C07305=1131.098,83.336,-54.639,179.925,7.711,149.479
C07306=1131.094,83.586,-54.656,179.926,7.715,149.480
C07307=1131.089,83.835,-54.674,179.927,7.718,149.480
C07308=1131.084,84.085,-54.691,179.929,7.722,149.481
C07309=1131.079,84.334,-54.709,179.930,7.726,149.481
C07310=1131.075,84.583,-54.727,179.932,7.730,149.482
C07311=1131.069,84.833,-54.744,179.932,7.734,149.482
C07312=1131.065,85.082,-54.762,179.934,7.738,149.483
C07313=1131.059,85.332,-54.779,179.935,7.742,149.483
C07314=1131.055,85.580,-54.796,179.937,7.745,149.483
C07315=1131.050,85.830,-54.814,179.938,7.749,149.484
C07316=1131.045,86.079,-54.832,179.939,7.753,149.485
C07317=1131.040,86.329,-54.850,179.941,7.757,149.485
C07318=1131.035,86.578,-54.867,179.942,7.761,149.486
C07319=1131.031,86.827,-54.884,179.943,7.765,149.486
C07320=1131.026,87.076,-54.902,179.945,7.769,149.486
C07321=1131.021,87.326,-54.920,179.947,7.773,149.487
C07322=1131.016,87.575,-54.938,179.947,7.776,149.487
C07323=1131.011,87.825,-54.955,179.949,7.780,149.488
C07324=1131.006,88.074,-54.973,179.950,7.784,149.488
C07325=1131.001,88.324,-54.991,179.952,7.788,149.489
C07326=1130.996,88.572,-55.008,179.954,7.792,149.489
C07327=1130.992,88.822,-55.026,179.955,7.796,149.490
C07328=1130.984,89.194,-55.053,179.957,7.802,149.490
C07329=1130.977,89.567,-55.079,179.959,7.808,149.491
C07330=1130.969,89.939,-55.106,179.962,7.814,149.492
C07331=1130.962,90.311,-55.132,179.964,7.819,149.492
C07332=1130.958,90.561,-55.150,179.966,7.823,149.493
C07333=1130.952,90.811,-55.167,179.967,7.827,149.493
C07334=1130.948,91.060,-55.185,179.969,7.831,149.494
C07335=1130.943,91.309,-55.203,179.971,7.835,149.494
C07336=1130.938,91.558,-55.221,179.972,7.839,149.495
C07337=1130.933,91.807,-55.239,179.974,7.843,149.495
C07338=1130.928,92.056,-55.257,179.975,7.847,149.495
C07339=1130.923,92.306,-55.275,179.977,7.851,149.496
C07340=1130.918,92.555,-55.293,179.979,7.854,149.496
C07341=1130.913,92.804,-55.311,179.980,7.858,149.497
C07342=1130.908,93.054,-55.329,179.982,7.863,149.497
C07343=1130.904,93.304,-55.347,179.984,7.867,149.498
C07344=1130.899,93.553,-55.365,179.986,7.871,149.498
C07345=1130.894,93.802,-55.383,179.987,7.875,149.498
C07346=1130.889,94.051,-55.401,179.989,7.879,149.499
C07347=1130.884,94.300,-55.419,179.990,7.882,149.499
C07348=1130.878,94.550,-55.437,179.992,7.886,149.500
C07349=1130.873,94.799,-55.455,179.994,7.891,149.500
C07350=1130.869,95.049,-55.474,179.996,7.895,149.500
C07351=1130.864,95.298,-55.492,179.998,7.898,149.501
C07352=1130.859,95.547,-55.510,180.000,7.902,149.501
C07353=1130.854,95.796,-55.528,-179.999,7.906,149.502
C07354=1130.850,96.045,-55.546,-179.997,7.911,149.502
C07355=1130.845,96.294,-55.564,-179.995,7.914,149.502
C07356=1130.841,96.544,-55.583,-179.993,7.918,149.503
C07357=1130.835,96.793,-55.601,-179.991,7.922,149.503
C07358=1130.830,97.043,-55.619,-179.989,7.927,149.503
C07359=1130.825,97.292,-55.637,-179.987,7.930,149.504
C07360=1130.820,97.541,-55.655,-179.986,7.934,149.504
C07361=1130.816,97.791,-55.673,-179.984,7.938,149.505
C07362=1130.811,98.039,-55.692,-179.981,7.942,149.505
C07363=1130.806,98.289,-55.711,-179.980,7.946,149.505
C07364=1130.801,98.538,-55.729,-179.978,7.950,149.506
C07365=1130.796,98.788,-55.747,-179.975,7.954,149.506
C07366=1130.791,99.037,-55.765,-179.974,7.958,149.506
C07367=1130.787,99.286,-55.784,-179.972,7.962,149.507
C07368=1130.781,99.535,-55.802,-179.969,7.967,149.507
C07369=1130.777,99.785,-55.821,-179.968,7.970,149.507
C07370=1130.772,100.034,-55.839,-179.966,7.974,149.508
C07371=1130.767,100.283,-55.857,-179.964,7.979,149.508
C07372=1130.762,100.532,-55.876,-179.962,7.982,149.508
C07373=1130.757,100.782,-55.894,-179.959,7.987,149.509
C07374=1130.753,101.031,-55.913,-179.957,7.990,149.509
C07375=1130.747,101.280,-55.932,-179.956,7.994,149.509
C07376=1130.743,101.530,-55.950,-179.953,7.998,149.509
C07377=1130.738,101.779,-55.969,-179.951,8.002,149.510
C07378=1130.733,102.028,-55.987,-179.949,8.007,149.510
C07379=1130.728,102.277,-56.005,-179.947,8.010,149.510
C07380=1130.724,102.492,-56.022,-179.945,8.014,149.511
C07381=1130.720,102.707,-56.038,-179.943,8.018,149.511
C07382=1130.716,102.923,-56.053,-179.941,8.021,149.511
C07383=1130.711,103.137,-56.070,-179.939,8.025,149.511
C07384=1130.707,103.352,-56.085,-179.937,8.028,149.512
C07385=1130.703,103.567,-56.102,-179.935,8.031,149.512
C07386=1130.699,103.782,-56.118,-179.933,8.034,149.512
C07387=1130.695,103.997,-56.134,-179.932,8.038,149.512
C07388=1130.690,104.246,-56.154,-179.929,8.042,149.513
C07389=1130.685,104.495,-56.171,-179.927,8.046,149.513
C07390=1130.681,104.745,-56.191,-179.924,8.050,149.513
C07391=1130.675,104.994,-56.209,-179.923,8.054,149.514
C07392=1130.670,105.243,-56.228,-179.920,8.058,149.514
C07393=1130.665,105.493,-56.247,-179.918,8.062,149.514
C07394=1130.661,105.741,-56.265,-179.915,8.066,149.514
C07395=1130.656,105.992,-56.284,-179.912,8.070,149.514
C07396=1130.651,106.240,-56.303,-179.910,8.074,149.515
C07397=1130.646,106.490,-56.323,-179.908,8.078,149.515
C07398=1130.642,106.739,-56.341,-179.906,8.082,149.515
C07399=1130.636,106.988,-56.360,-179.903,8.086,149.516
C07400=1130.632,107.237,-56.379,-179.901,8.091,149.516
C07401=1130.627,107.487,-56.398,-179.899,8.094,149.516
C07402=1130.623,107.736,-56.417,-179.896,8.098,149.516
C07403=1130.617,107.985,-56.436,-179.894,8.102,149.516
C07404=1130.613,108.235,-56.454,-179.891,8.106,149.517
C07405=1130.608,108.483,-56.474,-179.888,8.110,149.517
C07406=1130.603,108.733,-56.493,-179.886,8.114,149.517
C07407=1130.598,108.982,-56.512,-179.883,8.118,149.517
C07408=1130.593,109.232,-56.531,-179.881,8.122,149.517
C07409=1130.588,109.480,-56.550,-179.879,8.126,149.517
C07410=1130.584,109.730,-56.569,-179.876,8.130,149.518
C07411=1130.579,109.978,-56.588,-179.873,8.134,149.518
C07412=1130.574,110.228,-56.608,-179.871,8.139,149.518
C07413=1130.569,110.477,-56.627,-179.868,8.142,149.518
C07414=1130.565,110.727,-56.645,-179.865,8.146,149.518
C07415=1130.559,110.976,-56.665,-179.863,8.149,149.519
C07416=1130.555,111.225,-56.684,-179.861,8.153,149.519
C07417=1130.550,111.474,-56.703,-179.859,8.156,149.519
C07418=1130.545,111.723,-56.723,-179.858,8.160,149.519
C07419=1130.540,111.972,-56.742,-179.856,8.164,149.520
C07420=1130.535,112.222,-56.762,-179.853,8.167,149.520
C07421=1130.531,112.471,-56.781,-179.851,8.171,149.520
C07422=1130.526,112.720,-56.800,-179.849,8.174,149.520
C07423=1130.521,112.969,-56.820,-179.848,8.178,149.521
C07424=1130.517,113.218,-56.838,-179.846,8.182,149.521
C07425=1130.512,113.468,-56.858,-179.844,8.185,149.521
C07426=1130.506,113.716,-56.877,-179.842,8.189,149.521
C07427=1130.502,113.966,-56.897,-179.839,8.192,149.522
C07428=1130.497,114.216,-56.916,-179.838,8.196,149.522
C07429=1130.492,114.464,-56.935,-179.836,8.200,149.522
C07430=1130.488,114.714,-56.955,-179.834,8.203,149.523
C07431=1130.482,114.963,-56.974,-179.832,8.207,149.523
C07432=1130.478,115.212,-56.994,-179.830,8.210,149.523
C07433=1130.473,115.462,-57.013,-179.828,8.214,149.523
C07434=1130.468,115.710,-57.032,-179.826,8.217,149.524
C07435=1130.463,115.960,-57.052,-179.824,8.221,149.524
C07436=1130.459,116.175,-57.069,-179.822,8.224,149.524
C07437=1130.455,116.389,-57.086,-179.821,8.226,149.524
C07438=1130.451,116.604,-57.103,-179.819,8.230,149.524
C07439=1130.447,116.820,-57.120,-179.817,8.233,149.525
C07440=1130.442,117.034,-57.136,-179.816,8.235,149.525
C07441=1130.438,117.249,-57.153,-179.814,8.239,149.525
C07442=1130.434,117.464,-57.170,-179.813,8.241,149.525
C07443=1130.430,117.679,-57.187,-179.811,8.244,149.526
C07444=1130.425,117.928,-57.207,-179.809,8.248,149.526
C07445=1130.421,118.176,-57.226,-179.807,8.251,149.526
C07446=1130.416,118.426,-57.246,-179.805,8.255,149.526
C07447=1130.411,118.675,-57.266,-179.803,8.259,149.527
C07448=1130.407,118.925,-57.285,-179.801,8.262,149.527
C07449=1130.402,119.173,-57.305,-179.800,8.265,149.527
C07450=1130.397,119.423,-57.325,-179.798,8.268,149.527
C07451=1130.392,119.672,-57.345,-179.796,8.272,149.528
C07452=1130.387,119.920,-57.365,-179.794,8.276,149.528
C07453=1130.382,120.170,-57.384,-179.792,8.279,149.528
C07454=1130.378,120.420,-57.404,-179.790,8.283,149.528
C07455=1130.373,120.669,-57.424,-179.788,8.285,149.529
C07456=1130.368,120.917,-57.444,-179.786,8.289,149.529
C07457=1130.363,121.167,-57.463,-179.785,8.293,149.529
C07458=1130.359,121.416,-57.484,-179.783,8.296,149.530
C07459=1130.354,121.666,-57.503,-179.781,8.300,149.530
C07460=1130.349,121.914,-57.522,-179.779,8.302,149.530
C07461=1130.344,122.163,-57.543,-179.777,8.306,149.530
C07462=1130.339,122.413,-57.563,-179.775,8.309,149.530
C07463=1130.335,122.662,-57.583,-179.773,8.313,149.531
C07464=1130.330,122.911,-57.603,-179.772,8.316,149.531
C07465=1130.325,123.160,-57.622,-179.770,8.320,149.531
C07466=1130.320,123.409,-57.642,-179.768,8.323,149.532
C07467=1130.316,123.659,-57.662,-179.766,8.327,149.532
C07468=1130.311,123.908,-57.682,-179.765,8.330,149.532
C07469=1130.307,124.157,-57.702,-179.763,8.333,149.532
C07470=1130.301,124.406,-57.722,-179.761,8.337,149.533
C07471=1130.297,124.655,-57.742,-179.759,8.339,149.533
C07472=1130.292,124.904,-57.763,-179.758,8.343,149.533
C07473=1130.287,125.154,-57.782,-179.756,8.347,149.533
C07474=1130.282,125.403,-57.803,-179.753,8.350,149.534
C07475=1130.278,125.652,-57.823,-179.752,8.353,149.534
C07476=1130.273,125.901,-57.842,-179.750,8.356,149.534
C07477=1130.268,126.150,-57.863,-179.748,8.360,149.535
C07478=1130.263,126.399,-57.882,-179.747,8.363,149.535
C07479=1130.259,126.648,-57.903,-179.745,8.366,149.535
C07480=1130.254,126.897,-57.924,-179.743,8.370,149.535
C07481=1130.249,127.147,-57.943,-179.742,8.373,149.536
C07482=1130.245,127.396,-57.964,-179.740,8.377,149.536
C07483=1130.239,127.645,-57.983,-179.738,8.380,149.536
C07484=1130.235,127.894,-58.003,-179.736,8.383,149.536
C07485=1130.230,128.143,-58.024,-179.735,8.387,149.537
C07486=1130.225,128.393,-58.044,-179.732,8.390,149.537
C07487=1130.220,128.642,-58.064,-179.731,8.393,149.537
C07488=1130.216,128.891,-58.085,-179.729,8.397,149.538
C07489=1130.212,129.139,-58.105,-179.727,8.400,149.538
C07490=1130.206,129.389,-58.125,-179.726,8.403,149.538
C07491=1130.202,129.638,-58.146,-179.724,8.406,149.538
C07492=1130.197,129.852,-58.163,-179.722,8.409,149.539
C07493=1130.193,130.067,-58.180,-179.721,8.412,149.539
C07494=1130.189,130.282,-58.198,-179.720,8.415,149.539
C07495=1130.185,130.497,-58.216,-179.718,8.418,149.539
C07496=1130.181,130.712,-58.233,-179.717,8.420,149.540
C07497=1130.177,130.927,-58.251,-179.715,8.424,149.540
C07498=1130.173,131.141,-58.268,-179.713,8.427,149.540
C07499=1130.169,131.356,-58.285,-179.712,8.429,149.540
C07500=1130.164,131.605,-58.306,-179.711,8.432,149.541
C07501=1130.159,131.854,-58.327,-179.709,8.436,149.541
C07502=1130.155,132.103,-58.347,-179.708,8.439,149.541
C07503=1130.150,132.352,-58.368,-179.706,8.443,149.542
C07504=1130.145,132.602,-58.388,-179.704,8.446,149.542
C07505=1130.140,132.851,-58.408,-179.702,8.449,149.542
C07506=1130.136,133.100,-58.429,-179.701,8.453,149.543
C07507=1130.131,133.349,-58.449,-179.699,8.455,149.543
C07508=1130.126,133.598,-58.470,-179.697,8.459,149.543
C07509=1130.122,133.847,-58.490,-179.696,8.462,149.543
C07510=1130.117,134.096,-58.511,-179.694,8.465,149.544
C07511=1130.112,134.345,-58.532,-179.693,8.469,149.544
C07512=1130.107,134.595,-58.553,-179.691,8.472,149.544
C07513=1130.102,134.843,-58.573,-179.689,8.475,149.544
C07514=1130.098,135.092,-58.593,-179.688,8.479,149.545
C07515=1130.093,135.342,-58.614,-179.686,8.482,149.545
C07516=1130.088,135.591,-58.635,-179.685,8.485,149.546
C07517=1130.083,135.840,-58.656,-179.683,8.489,149.546
C07518=1130.079,136.089,-58.676,-179.681,8.491,149.546
C07519=1130.074,136.338,-58.697,-179.680,8.495,149.546
C07520=1130.069,136.587,-58.717,-179.678,8.498,149.547
C07521=1130.065,136.836,-58.738,-179.677,8.502,149.547
C07522=1130.060,137.085,-58.759,-179.675,8.505,149.547
C07523=1130.055,137.334,-58.779,-179.674,8.508,149.548
C07524=1130.050,137.583,-58.800,-179.672,8.511,149.548
C07525=1130.046,137.832,-58.820,-179.670,8.515,149.548
C07526=1130.041,138.082,-58.842,-179.669,8.518,149.549
C07527=1130.037,138.331,-58.862,-179.667,8.521,149.549
C07528=1130.031,138.581,-58.883,-179.666,8.524,149.549
C07529=1130.027,138.830,-58.903,-179.664,8.528,149.550
C07530=1130.022,139.078,-58.925,-179.663,8.531,149.550
C07531=1130.018,139.327,-58.945,-179.661,8.534,149.550
C07532=1130.012,139.576,-58.966,-179.660,8.537,149.551
C07533=1130.008,139.825,-58.987,-179.658,8.541,149.551
C07534=1130.003,140.075,-59.008,-179.657,8.544,149.551
C07535=1129.998,140.324,-59.028,-179.655,8.548,149.552
C07536=1129.994,140.572,-59.050,-179.654,8.551,149.552
C07537=1129.989,140.822,-59.071,-179.652,8.554,149.552
C07538=1129.984,141.071,-59.091,-179.651,8.557,149.553
C07539=1129.979,141.320,-59.112,-179.650,8.560,149.553
C07540=1129.975,141.569,-59.133,-179.647,8.564,149.553
C07541=1129.970,141.818,-59.155,-179.646,8.567,149.554
C07542=1129.966,142.067,-59.175,-179.645,8.571,149.554
C07543=1129.960,142.316,-59.196,-179.643,8.573,149.554
C07544=1129.956,142.566,-59.217,-179.642,8.577,149.555
C07545=1129.952,142.814,-59.238,-179.640,8.580,149.555
C07546=1129.947,143.064,-59.259,-179.639,8.584,149.555
C07547=1129.941,143.313,-59.280,-179.638,8.587,149.556
C07548=1129.938,143.527,-59.298,-179.636,8.590,149.556
C07549=1129.933,143.742,-59.316,-179.635,8.593,149.557
C07550=1129.930,143.957,-59.334,-179.634,8.595,149.557
C07551=1129.926,144.171,-59.353,-179.632,8.598,149.557
C07552=1129.922,144.385,-59.371,-179.631,8.601,149.557
C07553=1129.918,144.600,-59.389,-179.630,8.604,149.558
C07554=1129.913,144.815,-59.408,-179.629,8.607,149.558
C07555=1129.909,145.030,-59.426,-179.627,8.610,149.558
C07556=1129.904,145.279,-59.446,-179.625,8.613,149.559
C07557=1129.900,145.528,-59.469,-179.623,8.618,149.559
C07558=1129.896,145.777,-59.489,-179.619,8.621,149.559
C07559=1129.890,146.026,-59.510,-179.617,8.626,149.559
C07560=1129.886,146.275,-59.532,-179.614,8.630,149.559
C07561=1129.881,146.524,-59.552,-179.611,8.634,149.559
C07562=1129.877,146.773,-59.574,-179.609,8.637,149.559
C07563=1129.872,147.023,-59.595,-179.606,8.642,149.560
C07564=1129.867,147.271,-59.617,-179.603,8.646,149.560
C07565=1129.862,147.520,-59.637,-179.600,8.650,149.560
C07566=1129.858,147.770,-59.659,-179.598,8.653,149.560
C07567=1129.853,148.019,-59.680,-179.595,8.657,149.560
C07568=1129.848,148.267,-59.702,-179.592,8.661,149.560
C07569=1129.843,148.517,-59.723,-179.589,8.666,149.561
C07570=1129.839,148.766,-59.745,-179.587,8.669,149.561
C07571=1129.834,149.014,-59.766,-179.584,8.673,149.561
C07572=1129.829,149.264,-59.787,-179.582,8.677,149.561
C07573=1129.825,149.513,-59.809,-179.579,8.680,149.561
C07574=1129.820,149.762,-59.830,-179.576,8.685,149.561
C07575=1129.815,150.011,-59.851,-179.573,8.689,149.561
C07576=1129.811,150.260,-59.874,-179.571,8.692,149.562
C07577=1129.806,150.509,-59.895,-179.568,8.696,149.562
C07578=1129.801,150.758,-59.916,-179.566,8.699,149.562
C07579=1129.797,151.007,-59.938,-179.563,8.703,149.562
C07580=1129.792,151.256,-59.959,-179.560,8.708,149.562
C07581=1129.787,151.504,-59.981,-179.557,8.711,149.562
C07582=1129.783,151.754,-60.002,-179.555,8.715,149.563
C07583=1129.778,152.003,-60.024,-179.552,8.718,149.563
C07584=1129.773,152.252,-60.046,-179.550,8.722,149.563
C07585=1129.769,152.501,-60.068,-179.547,8.725,149.563
C07586=1129.764,152.750,-60.089,-179.544,8.730,149.563
C07587=1129.759,153.000,-60.111,-179.542,8.733,149.563
C07588=1129.755,153.248,-60.132,-179.539,8.737,149.563
C07589=1129.750,153.497,-60.154,-179.537,8.740,149.563
C07590=1129.745,153.746,-60.176,-179.534,8.744,149.564
C07591=1129.741,153.995,-60.198,-179.531,8.747,149.564
C07592=1129.736,154.244,-60.220,-179.528,8.751,149.564
C07593=1129.731,154.493,-60.242,-179.526,8.755,149.564
C07594=1129.727,154.741,-60.263,-179.523,8.759,149.564
C07595=1129.722,154.991,-60.285,-179.521,8.762,149.564
C07596=1129.717,155.240,-60.308,-179.518,8.765,149.564
C07597=1129.712,155.489,-60.330,-179.515,8.769,149.564
C07598=1129.708,155.738,-60.351,-179.513,8.773,149.564
C07599=1129.703,155.987,-60.373,-179.510,8.777,149.564
C07600=1129.698,156.236,-60.395,-179.508,8.780,149.565
C07601=1129.694,156.485,-60.417,-179.505,8.783,149.565
C07602=1129.689,156.734,-60.439,-179.502,8.787,149.565
C07603=1129.685,156.983,-60.461,-179.500,8.791,149.565
C07604=1129.681,157.198,-60.479,-179.498,8.794,149.565
C07605=1129.676,157.412,-60.498,-179.496,8.796,149.565
C07606=1129.672,157.626,-60.517,-179.494,8.799,149.565
C07607=1129.669,157.841,-60.537,-179.491,8.803,149.565
C07608=1129.665,158.056,-60.555,-179.489,8.806,149.565
C07609=1129.660,158.270,-60.574,-179.487,8.808,149.565
C07610=1129.657,158.485,-60.594,-179.485,8.812,149.566
C07611=1129.653,158.699,-60.613,-179.482,8.815,149.566
C07612=1129.647,158.948,-60.635,-179.479,8.818,149.566
C07613=1129.643,159.198,-60.657,-179.477,8.821,149.566
C07614=1129.638,159.446,-60.679,-179.475,8.824,149.566
C07615=1129.634,159.695,-60.701,-179.472,8.828,149.566
C07616=1129.629,159.945,-60.724,-179.469,8.831,149.566
C07617=1129.624,160.193,-60.746,-179.467,8.835,149.566
C07618=1129.620,160.443,-60.768,-179.465,8.838,149.566
C07619=1129.615,160.691,-60.790,-179.462,8.841,149.566
C07620=1129.610,160.940,-60.813,-179.460,8.845,149.566
C07621=1129.606,161.190,-60.835,-179.457,8.848,149.567
C07622=1129.601,161.438,-60.857,-179.454,8.851,149.567
C07623=1129.597,161.687,-60.880,-179.452,8.855,149.567
C07624=1129.592,161.936,-60.902,-179.450,8.858,149.567
C07625=1129.587,162.185,-60.924,-179.447,8.861,149.567
C07626=1129.583,162.434,-60.947,-179.445,8.864,149.567
C07627=1129.578,162.683,-60.969,-179.443,8.868,149.567
C07628=1129.574,162.932,-60.991,-179.439,8.872,149.567
C07629=1129.568,163.181,-61.014,-179.437,8.875,149.567
C07630=1129.564,163.430,-61.036,-179.434,8.878,149.567
C07631=1129.560,163.679,-61.059,-179.432,8.881,149.567
C07632=1129.555,163.928,-61.081,-179.430,8.884,149.567
C07633=1129.551,164.176,-61.104,-179.427,8.888,149.568
C07634=1129.546,164.426,-61.126,-179.425,8.891,149.568
C07635=1129.541,164.675,-61.148,-179.423,8.894,149.568
C07636=1129.537,164.923,-61.171,-179.420,8.897,149.568
C07637=1129.532,165.173,-61.193,-179.418,8.900,149.568
C07638=1129.527,165.421,-61.216,-179.415,8.903,149.568
C07639=1129.522,165.670,-61.239,-179.413,8.907,149.568
C07640=1129.518,165.919,-61.261,-179.410,8.910,149.568
C07641=1129.513,166.168,-61.285,-179.408,8.913,149.568
C07642=1129.509,166.417,-61.306,-179.405,8.916,149.568
C07643=1129.505,166.666,-61.329,-179.403,8.919,149.568
C07644=1129.500,166.915,-61.352,-179.401,8.923,149.568
C07645=1129.495,167.163,-61.374,-179.398,8.926,149.569
C07646=1129.490,167.412,-61.397,-179.396,8.929,149.569
C07647=1129.485,167.662,-61.420,-179.393,8.932,149.569
C07648=1129.481,167.911,-61.443,-179.391,8.936,149.569
C07649=1129.476,168.160,-61.465,-179.389,8.938,149.569
C07650=1129.472,168.408,-61.488,-179.387,8.941,149.569
C07651=1129.467,168.657,-61.511,-179.384,8.944,149.569
C07652=1129.463,168.906,-61.534,-179.382,8.948,149.569
C07653=1129.458,169.155,-61.556,-179.380,8.951,149.569
C07654=1129.454,169.404,-61.579,-179.377,8.954,149.569
C07655=1129.449,169.653,-61.602,-179.375,8.957,149.569
C07656=1129.444,169.903,-61.625,-179.372,8.961,149.569
C07657=1129.439,170.151,-61.648,-179.371,8.963,149.570
C07658=1129.435,170.400,-61.671,-179.368,8.966,149.570
C07659=1129.431,170.648,-61.694,-179.365,8.969,149.570
C07660=1129.426,170.863,-61.713,-179.364,8.972,149.570
C07661=1129.422,171.078,-61.733,-179.361,8.975,149.570
C07662=1129.418,171.292,-61.753,-179.360,8.977,149.570
C07663=1129.414,171.507,-61.773,-179.358,8.980,149.570
C07664=1129.410,171.721,-61.792,-179.355,8.983,149.570
C07665=1129.406,171.935,-61.812,-179.354,8.985,149.570
C07666=1129.402,172.149,-61.832,-179.352,8.988,149.570
C07667=1129.398,172.364,-61.852,-179.350,8.990,149.570
C07668=1129.394,172.613,-61.875,-179.347,8.993,149.570
C07669=1129.389,172.862,-61.898,-179.345,8.997,149.571
C07670=1129.385,173.111,-61.921,-179.343,9.000,149.571
C07671=1129.379,173.360,-61.944,-179.341,9.002,149.571
C07672=1129.375,173.609,-61.967,-179.338,9.005,149.571
C07673=1129.371,173.858,-61.990,-179.336,9.009,149.571
C07674=1129.366,174.107,-62.014,-179.334,9.011,149.571
C07675=1129.362,174.355,-62.036,-179.332,9.014,149.571
C07676=1129.357,174.604,-62.060,-179.330,9.018,149.571
C07677=1129.353,174.853,-62.083,-179.327,9.021,149.571
C07678=1129.347,175.102,-62.106,-179.325,9.023,149.571
C07679=1129.343,175.350,-62.129,-179.323,9.026,149.571
C07680=1129.339,175.599,-62.152,-179.321,9.030,149.571
C07681=1129.334,175.848,-62.176,-179.319,9.032,149.572
C07682=1129.329,176.098,-62.199,-179.316,9.035,149.572
C07683=1129.325,176.347,-62.222,-179.314,9.038,149.572
C07684=1129.321,176.595,-62.245,-179.312,9.041,149.572
C07685=1129.316,176.844,-62.268,-179.310,9.044,149.572
C07686=1129.311,177.093,-62.292,-179.308,9.047,149.572
C07687=1129.307,177.342,-62.315,-179.306,9.050,149.572
C07688=1129.302,177.591,-62.339,-179.303,9.053,149.572
C07689=1129.298,177.839,-62.362,-179.302,9.056,149.572
C07690=1129.293,178.089,-62.385,-179.299,9.059,149.572
C07691=1129.288,178.337,-62.408,-179.297,9.062,149.573
C07692=1129.283,178.586,-62.432,-179.295,9.064,149.573
C07693=1129.279,178.835,-62.455,-179.293,9.068,149.573
C07694=1129.274,179.084,-62.478,-179.291,9.070,149.573
C07695=1129.270,179.332,-62.502,-179.288,9.074,149.573
C07696=1129.265,179.581,-62.526,-179.285,9.077,149.573
C07697=1129.261,179.830,-62.549,-179.282,9.081,149.573
C07698=1129.256,180.079,-62.572,-179.280,9.084,149.573
C07699=1129.252,180.328,-62.596,-179.276,9.087,149.573
C07700=1129.247,180.577,-62.619,-179.273,9.091,149.573
C07701=1129.243,180.826,-62.643,-179.270,9.094,149.573
C07702=1129.238,181.075,-62.666,-179.267,9.098,149.573
C07703=1129.233,181.323,-62.690,-179.264,9.101,149.573
C07704=1129.229,181.572,-62.713,-179.262,9.104,149.573
C07705=1129.224,181.821,-62.737,-179.258,9.108,149.573
C07706=1129.220,182.070,-62.761,-179.256,9.111,149.573
C07707=1129.216,182.319,-62.785,-179.253,9.114,149.573
C07708=1129.211,182.568,-62.808,-179.249,9.117,149.573
C07709=1129.206,182.817,-62.832,-179.247,9.120,149.573
C07710=1129.202,183.066,-62.855,-179.244,9.124,149.573
C07711=1129.197,183.314,-62.880,-179.241,9.126,149.573
C07712=1129.193,183.563,-62.903,-179.238,9.130,149.573
C07713=1129.188,183.812,-62.927,-179.236,9.133,149.573
C07714=1129.184,184.061,-62.950,-179.233,9.136,149.573
C07715=1129.179,184.309,-62.974,-179.230,9.139,149.573
C07716=1129.175,184.524,-62.995,-179.228,9.141,149.573
C07717=1129.171,184.738,-63.016,-179.226,9.145,149.573
C07718=1129.167,184.953,-63.036,-179.224,9.147,149.573
C07719=1129.163,185.167,-63.056,-179.221,9.150,149.573
C07720=1129.159,185.382,-63.077,-179.219,9.152,149.572
C07721=1129.156,185.596,-63.098,-179.217,9.155,149.573
C07722=1129.151,185.809,-63.118,-179.215,9.157,149.573
C07723=1129.147,186.024,-63.139,-179.213,9.160,149.573
C07724=1129.143,186.273,-63.163,-179.210,9.163,149.573
C07725=1129.138,186.521,-63.187,-179.208,9.166,149.573
C07726=1129.134,186.770,-63.210,-179.205,9.169,149.573
C07727=1129.130,187.020,-63.234,-179.203,9.171,149.573
C07728=1129.125,187.268,-63.259,-179.200,9.174,149.573
C07729=1129.120,187.517,-63.282,-179.198,9.177,149.573
C07730=1129.116,187.766,-63.306,-179.195,9.180,149.573
C07731=1129.111,188.014,-63.331,-179.193,9.183,149.573
C07732=1129.106,188.263,-63.354,-179.191,9.186,149.573
C07733=1129.102,188.513,-63.379,-179.189,9.188,149.573
C07734=1129.098,188.761,-63.403,-179.186,9.191,149.573
C07735=1129.093,189.010,-63.426,-179.184,9.194,149.573
C07736=1129.088,189.259,-63.450,-179.182,9.197,149.573
C07737=1129.083,189.507,-63.475,-179.180,9.200,149.573
C07738=1129.079,189.756,-63.499,-179.178,9.202,149.573
C07739=1129.075,190.005,-63.523,-179.176,9.206,149.573
C07740=1129.070,190.254,-63.547,-179.174,9.208,149.573
C07741=1129.065,190.503,-63.572,-179.172,9.210,149.573
C07742=1129.061,190.751,-63.596,-179.169,9.213,149.573
C07743=1129.057,191.001,-63.619,-179.167,9.216,149.573
C07744=1129.052,191.249,-63.644,-179.165,9.218,149.573
C07745=1129.047,191.498,-63.668,-179.163,9.221,149.574
C07746=1129.043,191.746,-63.692,-179.161,9.224,149.574
C07747=1129.038,191.995,-63.717,-179.160,9.226,149.574
C07748=1129.034,192.244,-63.741,-179.158,9.229,149.574
C07749=1129.030,192.492,-63.765,-179.156,9.232,149.574
C07750=1129.024,192.742,-63.789,-179.154,9.234,149.574
C07751=1129.020,192.991,-63.814,-179.152,9.237,149.574
C07752=1129.016,193.239,-63.838,-179.150,9.239,149.574
C07753=1129.011,193.488,-63.863,-179.149,9.242,149.575
C07754=1129.006,193.736,-63.887,-179.147,9.244,149.575
C07755=1129.003,193.986,-63.911,-179.145,9.247,149.575
C07756=1128.998,194.234,-63.936,-179.144,9.249,149.575
C07757=1128.993,194.483,-63.960,-179.142,9.252,149.575
C07758=1128.988,194.731,-63.985,-179.140,9.254,149.575
C07759=1128.984,194.981,-64.009,-179.139,9.257,149.575
C07760=1128.980,195.229,-64.033,-179.137,9.260,149.576
C07761=1128.975,195.478,-64.058,-179.135,9.262,149.576
C07762=1128.971,195.727,-64.082,-179.134,9.265,149.576
C07763=1128.966,195.976,-64.107,-179.132,9.268,149.576
C07764=1128.961,196.224,-64.131,-179.131,9.270,149.576
C07765=1128.957,196.473,-64.156,-179.127,9.274,149.576
C07766=1128.952,196.722,-64.180,-179.124,9.277,149.576
C07767=1128.947,196.970,-64.205,-179.120,9.282,149.576
C07768=1128.943,197.220,-64.229,-179.116,9.285,149.576
C07769=1128.939,197.468,-64.253,-179.112,9.289,149.576
C07770=1128.934,197.717,-64.278,-179.108,9.293,149.576
C07771=1128.930,197.966,-64.302,-179.104,9.296,149.575
C07772=1128.926,198.180,-64.324,-179.101,9.300,149.575
C07773=1128.922,198.395,-64.345,-179.098,9.303,149.575
C07774=1128.918,198.608,-64.366,-179.095,9.305,149.575
C07775=1128.914,198.822,-64.388,-179.092,9.309,149.575
C07776=1128.910,199.037,-64.409,-179.089,9.312,149.575
C07777=1128.907,199.250,-64.430,-179.085,9.315,149.575
C07778=1128.902,199.465,-64.451,-179.082,9.318,149.574
C07779=1128.898,199.679,-64.473,-179.079,9.321,149.574
C07780=1128.895,199.928,-64.497,-179.075,9.324,149.574
C07781=1128.890,200.177,-64.523,-179.072,9.328,149.574
C07782=1128.885,200.426,-64.548,-179.068,9.331,149.574
C07783=1128.881,200.674,-64.572,-179.065,9.335,149.574
C07784=1128.876,200.922,-64.597,-179.062,9.337,149.574
C07785=1128.872,201.172,-64.622,-179.058,9.341,149.573
C07786=1128.867,201.420,-64.646,-179.055,9.344,149.573
C07787=1128.863,201.669,-64.672,-179.052,9.347,149.573
C07788=1128.858,201.918,-64.696,-179.048,9.351,149.573
C07789=1128.854,202.167,-64.721,-179.045,9.353,149.573
C07790=1128.849,202.415,-64.747,-179.042,9.357,149.573
C07791=1128.845,202.665,-64.772,-179.039,9.360,149.573
C07792=1128.840,202.912,-64.796,-179.035,9.363,149.572
C07793=1128.836,203.162,-64.821,-179.032,9.366,149.572
C07794=1128.831,203.410,-64.847,-179.028,9.369,149.572
C07795=1128.827,203.659,-64.871,-179.026,9.373,149.572
C07796=1128.822,203.907,-64.897,-179.023,9.375,149.572
C07797=1128.818,204.156,-64.922,-179.020,9.378,149.572
C07798=1128.813,204.405,-64.947,-179.017,9.381,149.572
C07799=1128.809,204.654,-64.972,-179.013,9.384,149.572
C07800=1128.804,204.902,-64.997,-179.011,9.387,149.572
C07801=1128.800,205.151,-65.023,-179.008,9.390,149.571
C07802=1128.796,205.400,-65.048,-179.005,9.393,149.571
C07803=1128.791,205.648,-65.073,-179.002,9.396,149.571
C07804=1128.786,205.898,-65.098,-179.000,9.399,149.571
C07805=1128.782,206.146,-65.123,-178.997,9.401,149.571
C07806=1128.777,206.394,-65.149,-178.994,9.403,149.571
C07807=1128.773,206.643,-65.173,-178.992,9.407,149.571
C07808=1128.769,206.892,-65.199,-178.989,9.409,149.571
C07809=1128.764,207.140,-65.225,-178.986,9.412,149.571
C07810=1128.759,207.389,-65.249,-178.983,9.415,149.571
C07811=1128.755,207.638,-65.275,-178.981,9.417,149.571
C07812=1128.750,207.886,-65.301,-178.979,9.421,149.571
C07813=1128.746,208.135,-65.326,-178.976,9.423,149.571
C07814=1128.742,208.384,-65.351,-178.974,9.426,149.571
C07815=1128.737,208.632,-65.377,-178.972,9.429,149.571
C07816=1128.732,208.881,-65.402,-178.969,9.431,149.571
C07817=1128.728,209.130,-65.428,-178.967,9.434,149.571
C07818=1128.724,209.378,-65.453,-178.965,9.436,149.571
C07819=1128.720,209.627,-65.478,-178.962,9.439,149.571
C07820=1128.715,209.875,-65.503,-178.960,9.442,149.571
C07821=1128.711,210.124,-65.529,-178.959,9.444,149.571
C07822=1128.706,210.373,-65.555,-178.956,9.447,149.571
C07823=1128.702,210.621,-65.580,-178.954,9.449,149.571
C07824=1128.697,210.870,-65.606,-178.952,9.452,149.571
C07825=1128.693,211.119,-65.631,-178.950,9.454,149.571
C07826=1128.688,211.367,-65.656,-178.948,9.457,149.571
C07827=1128.684,211.616,-65.682,-178.946,9.459,149.571
C07828=1128.680,211.830,-65.705,-178.945,9.461,149.571
C07829=1128.676,212.044,-65.727,-178.943,9.464,149.571
C07830=1128.672,212.259,-65.749,-178.941,9.466,149.572
C07831=1128.668,212.473,-65.771,-178.940,9.468,149.572
C07832=1128.665,212.686,-65.793,-178.939,9.470,149.572
C07833=1128.660,212.901,-65.815,-178.937,9.473,149.572
C07834=1128.657,213.115,-65.837,-178.936,9.475,149.572
C07835=1128.653,213.330,-65.859,-178.934,9.477,149.572
C07836=1128.648,213.578,-65.885,-178.932,9.480,149.572
C07837=1128.644,213.827,-65.910,-178.931,9.482,149.573
C07838=1128.640,214.075,-65.936,-178.929,9.485,149.573
C07839=1128.635,214.323,-65.961,-178.927,9.488,149.573
C07840=1128.631,214.572,-65.987,-178.925,9.490,149.573
C07841=1128.626,214.821,-66.013,-178.923,9.493,149.573
C07842=1128.622,215.070,-66.039,-178.921,9.496,149.573
C07843=1128.617,215.318,-66.065,-178.919,9.499,149.573
C07844=1128.613,215.566,-66.091,-178.918,9.501,149.574
C07845=1128.608,215.815,-66.117,-178.915,9.504,149.574
C07846=1128.604,216.064,-66.143,-178.914,9.507,149.574
C07847=1128.599,216.312,-66.168,-178.911,9.510,149.574
C07848=1128.595,216.561,-66.194,-178.909,9.513,149.574
C07849=1128.591,216.810,-66.220,-178.907,9.516,149.574
C07850=1128.586,217.059,-66.246,-178.905,9.519,149.574
C07851=1128.582,217.308,-66.272,-178.903,9.521,149.574
C07852=1128.577,217.556,-66.297,-178.901,9.525,149.575
C07853=1128.573,217.804,-66.324,-178.898,9.528,149.575
C07854=1128.569,218.053,-66.349,-178.896,9.530,149.575
C07855=1128.565,218.302,-66.375,-178.894,9.534,149.575
C07856=1128.560,218.551,-66.401,-178.892,9.537,149.575
C07857=1128.555,218.799,-66.427,-178.889,9.540,149.575
C07858=1128.551,219.047,-66.453,-178.887,9.543,149.575
C07859=1128.547,219.296,-66.479,-178.885,9.545,149.575
C07860=1128.542,219.545,-66.505,-178.882,9.549,149.575
C07861=1128.537,219.794,-66.531,-178.880,9.552,149.575
C07862=1128.533,220.041,-66.557,-178.877,9.555,149.576
C07863=1128.529,220.290,-66.583,-178.875,9.558,149.576
C07864=1128.524,220.539,-66.609,-178.872,9.561,149.576
C07865=1128.520,220.787,-66.636,-178.870,9.564,149.576
C07866=1128.516,221.036,-66.661,-178.867,9.568,149.576
C07867=1128.511,221.285,-66.687,-178.864,9.571,149.576
C07868=1128.507,221.533,-66.714,-178.862,9.575,149.576
C07869=1128.502,221.782,-66.740,-178.859,9.578,149.576
C07870=1128.498,222.030,-66.765,-178.857,9.581,149.576
C07871=1128.493,222.279,-66.792,-178.854,9.584,149.576
C07872=1128.489,222.528,-66.818,-178.851,9.587,149.576
C07873=1128.484,222.776,-66.845,-178.848,9.591,149.576
C07874=1128.480,223.025,-66.871,-178.845,9.594,149.576
C07875=1128.476,223.274,-66.897,-178.842,9.598,149.576
C07876=1128.471,223.522,-66.924,-178.839,9.600,149.576
C07877=1128.467,223.771,-66.950,-178.837,9.603,149.576
C07878=1128.463,224.019,-66.976,-178.834,9.607,149.576
C07879=1128.458,224.268,-67.002,-178.831,9.610,149.576
C07880=1128.453,224.516,-67.029,-178.828,9.614,149.576
C07881=1128.448,224.765,-67.055,-178.825,9.617,149.576
C07882=1128.445,225.013,-67.081,-178.821,9.621,149.576
C07883=1128.440,225.262,-67.108,-178.819,9.624,149.576
C07884=1128.436,225.477,-67.131,-178.816,9.626,149.576
C07885=1128.433,225.690,-67.153,-178.813,9.629,149.576
C07886=1128.429,225.904,-67.176,-178.810,9.632,149.576
C07887=1128.425,226.118,-67.199,-178.808,9.635,149.576
C07888=1128.421,226.332,-67.222,-178.805,9.638,149.576
C07889=1128.418,226.546,-67.245,-178.802,9.641,149.576
C07890=1128.414,226.760,-67.268,-178.800,9.644,149.576
C07891=1128.410,226.973,-67.291,-178.796,9.647,149.576
C07892=1128.405,227.222,-67.317,-178.793,9.650,149.576
C07893=1128.401,227.471,-67.343,-178.790,9.654,149.576
C07894=1128.396,227.719,-67.370,-178.786,9.658,149.576
C07895=1128.392,227.967,-67.397,-178.783,9.661,149.575
C07896=1128.387,228.216,-67.423,-178.779,9.665,149.575
C07897=1128.384,228.465,-67.450,-178.776,9.667,149.575
C07898=1128.379,228.714,-67.477,-178.773,9.671,149.575
C07899=1128.375,228.962,-67.504,-178.769,9.674,149.575
C07900=1128.371,229.211,-67.530,-178.765,9.678,149.575
C07901=1128.366,229.460,-67.557,-178.762,9.681,149.575
C07902=1128.361,229.708,-67.584,-178.758,9.685,149.574
C07903=1128.357,229.956,-67.610,-178.754,9.688,149.574
C07904=1128.353,230.205,-67.638,-178.751,9.692,149.574
C07905=1128.348,230.453,-67.665,-178.747,9.695,149.574
C07906=1128.344,230.701,-67.691,-178.743,9.698,149.574
C07907=1128.339,230.950,-67.718,-178.739,9.702,149.574
C07908=1128.335,231.198,-67.745,-178.736,9.705,149.574
C07909=1128.331,231.447,-67.772,-178.733,9.708,149.573
C07910=1128.327,231.696,-67.799,-178.729,9.712,149.573
C07911=1128.322,231.944,-67.826,-178.725,9.715,149.573
C07912=1128.317,232.193,-67.853,-178.722,9.718,149.573
C07913=1128.314,232.441,-67.880,-178.719,9.721,149.573
C07914=1128.309,232.689,-67.907,-178.716,9.724,149.573
C07915=1128.304,232.938,-67.934,-178.712,9.727,149.573
C07916=1128.300,233.187,-67.961,-178.709,9.730,149.572
C07917=1128.296,233.436,-67.988,-178.706,9.733,149.572
C07918=1128.292,233.684,-68.015,-178.703,9.736,149.572
C07919=1128.287,233.932,-68.042,-178.700,9.739,149.572
C07920=1128.283,234.180,-68.070,-178.697,9.742,149.572
C07921=1128.279,234.429,-68.097,-178.693,9.745,149.572
C07922=1128.274,234.678,-68.124,-178.690,9.748,149.571
C07923=1128.269,234.926,-68.151,-178.687,9.751,149.571
C07924=1128.265,235.175,-68.178,-178.684,9.753,149.571
C07925=1128.261,235.422,-68.205,-178.681,9.756,149.571
C07926=1128.257,235.672,-68.233,-178.678,9.759,149.571
C07927=1128.252,235.920,-68.260,-178.675,9.762,149.571
C07928=1128.248,236.169,-68.287,-178.673,9.765,149.571
C07929=1128.243,236.416,-68.315,-178.670,9.767,149.571
C07930=1128.239,236.666,-68.342,-178.667,9.770,149.571
C07931=1128.235,236.914,-68.369,-178.665,9.772,149.570
C07932=1128.230,237.163,-68.396,-178.662,9.775,149.570
C07933=1128.226,237.411,-68.424,-178.659,9.778,149.570
C07934=1128.221,237.660,-68.451,-178.656,9.780,149.570
C07935=1128.217,237.908,-68.479,-178.654,9.783,149.570
C07936=1128.212,238.156,-68.506,-178.651,9.785,149.570
C07937=1128.209,238.404,-68.533,-178.649,9.787,149.570
C07938=1128.205,238.653,-68.561,-178.646,9.791,149.570
C07939=1128.200,238.901,-68.588,-178.643,9.793,149.570
C07940=1128.196,239.115,-68.612,-178.641,9.795,149.570
C07941=1128.192,239.329,-68.635,-178.639,9.798,149.570
C07942=1128.188,239.543,-68.660,-178.637,9.799,149.570
C07943=1128.185,239.757,-68.683,-178.635,9.801,149.570
C07944=1128.181,239.970,-68.706,-178.633,9.803,149.570
C07945=1128.177,240.185,-68.731,-178.631,9.805,149.570
C07946=1128.174,240.399,-68.754,-178.629,9.808,149.570
C07947=1128.170,240.612,-68.777,-178.627,9.810,149.569
C07948=1128.165,240.861,-68.806,-178.625,9.812,149.570
C07949=1128.161,241.109,-68.833,-178.623,9.814,149.569
C07950=1128.156,241.358,-68.860,-178.621,9.816,149.569
C07951=1128.153,241.606,-68.888,-178.618,9.819,149.570
C07952=1128.148,241.855,-68.916,-178.616,9.821,149.569
C07953=1128.144,242.103,-68.943,-178.614,9.824,149.569
C07954=1128.140,242.351,-68.971,-178.612,9.826,149.570
C07955=1128.135,242.600,-68.999,-178.610,9.828,149.570
C07956=1128.131,242.848,-69.026,-178.608,9.831,149.570
C07957=1128.127,243.097,-69.054,-178.606,9.833,149.570
C07958=1128.122,243.345,-69.082,-178.605,9.835,149.570
C07959=1128.117,243.594,-69.109,-178.603,9.837,149.570
C07960=1128.113,243.842,-69.137,-178.601,9.839,149.570
C07961=1128.109,244.090,-69.165,-178.599,9.842,149.570
C07962=1128.105,244.339,-69.193,-178.598,9.844,149.570
C07963=1128.101,244.587,-69.220,-178.596,9.846,149.570
C07964=1128.096,244.835,-69.248,-178.594,9.848,149.570
C07965=1128.092,245.084,-69.276,-178.593,9.851,149.570
C07966=1128.087,245.332,-69.304,-178.591,9.853,149.570
C07967=1128.083,245.581,-69.332,-178.590,9.854,149.570
C07968=1128.079,245.829,-69.359,-178.588,9.857,149.571
C07969=1128.074,246.077,-69.387,-178.587,9.859,149.571
C07970=1128.070,246.326,-69.415,-178.586,9.861,149.571
C07971=1128.065,246.575,-69.443,-178.584,9.863,149.571
C07972=1128.061,246.823,-69.471,-178.583,9.866,149.571
C07973=1128.057,247.071,-69.499,-178.582,9.867,149.571
C07974=1128.053,247.320,-69.527,-178.580,9.870,149.572
C07975=1128.049,247.568,-69.554,-178.575,9.874,149.571
C07976=1128.044,247.816,-69.582,-178.569,9.879,149.571
C07977=1128.040,248.065,-69.610,-178.562,9.885,149.570
C07978=1128.035,248.313,-69.638,-178.555,9.890,149.570
C07979=1128.032,248.561,-69.666,-178.549,9.895,149.569
C07980=1128.027,248.810,-69.695,-178.544,9.899,149.569
C07981=1128.023,249.059,-69.722,-178.537,9.903,149.568
C07982=1128.018,249.307,-69.750,-178.532,9.908,149.568
C07983=1128.014,249.556,-69.779,-178.526,9.912,149.568
C07984=1128.009,249.803,-69.806,-178.521,9.916,149.567
C07985=1128.005,250.052,-69.835,-178.516,9.919,149.567
C07986=1128.000,250.300,-69.863,-178.512,9.923,149.566
C07987=1127.997,250.549,-69.891,-178.507,9.927,149.566
C07988=1127.993,250.797,-69.920,-178.503,9.930,149.566
C07989=1127.988,251.045,-69.948,-178.499,9.933,149.565
C07990=1127.984,251.294,-69.977,-178.495,9.936,149.565
C07991=1127.979,251.542,-70.005,-178.491,9.940,149.565
C07992=1127.975,251.791,-70.033,-178.488,9.942,149.565
C07993=1127.971,252.038,-70.061,-178.484,9.945,149.564
C07994=1127.966,252.287,-70.090,-178.482,9.948,149.564
C07995=1127.962,252.536,-70.118,-178.479,9.950,149.564
C07996=1127.959,252.749,-70.143,-178.477,9.951,149.564
C07997=1127.954,252.963,-70.167,-178.475,9.953,149.564
C07998=1127.951,253.176,-70.191,-178.473,9.955,149.564
C07999=1127.948,253.390,-70.216,-178.472,9.957,149.564
C08000=1127.944,253.604,-70.241,-178.470,9.958,149.564
C08001=1127.940,253.818,-70.265,-178.469,9.959,149.564
C08002=1127.936,254.032,-70.290,-178.468,9.961,149.564
C08003=1127.933,254.245,-70.314,-178.467,9.962,149.564
C08004=1127.928,254.493,-70.343,-178.466,9.964,149.564
C08005=1127.924,254.742,-70.371,-178.466,9.965,149.564
C08006=1127.920,254.990,-70.400,-178.466,9.966,149.564
C08007=1127.915,255.238,-70.429,-178.466,9.967,149.565
C08008=1127.911,255.487,-70.457,-178.466,9.967,149.565
C08009=1127.907,255.736,-70.486,-178.466,9.968,149.565
C08010=1127.903,255.983,-70.514,-178.467,9.969,149.565
C08011=1127.898,256.232,-70.543,-178.464,9.972,149.565
C08012=1127.894,256.480,-70.571,-178.461,9.975,149.565
C08013=1127.889,256.729,-70.599,-178.458,9.977,149.565
C08014=1127.886,256.977,-70.628,-178.455,9.981,149.565
C08015=1127.881,257.225,-70.657,-178.452,9.984,149.565
C08016=1127.876,257.474,-70.685,-178.449,9.987,149.565
C08017=1127.873,257.722,-70.714,-178.446,9.990,149.565
C08018=1127.868,257.970,-70.743,-178.443,9.992,149.565
C08019=1127.864,258.218,-70.771,-178.440,9.995,149.565
C08020=1127.860,258.467,-70.800,-178.436,9.999,149.565
C08021=1127.855,258.716,-70.829,-178.434,10.001,149.565
C08022=1127.851,258.963,-70.857,-178.431,10.004,149.564
C08023=1127.847,259.212,-70.886,-178.428,10.007,149.564
C08024=1127.843,259.460,-70.916,-178.424,10.010,149.564
C08025=1127.838,259.708,-70.943,-178.421,10.013,149.564
C08026=1127.834,259.956,-70.973,-178.417,10.016,149.564
C08027=1127.830,260.205,-71.002,-178.414,10.019,149.564
C08028=1127.826,260.453,-71.031,-178.411,10.022,149.564
C08029=1127.821,260.701,-71.059,-178.407,10.025,149.563
C08030=1127.817,260.949,-71.088,-178.404,10.028,149.563
C08031=1127.812,261.198,-71.117,-178.401,10.031,149.563
C08032=1127.809,261.446,-71.146,-178.397,10.035,149.563
C08033=1127.804,261.694,-71.174,-178.394,10.037,149.563
C08034=1127.800,261.943,-71.204,-178.390,10.041,149.563
C08035=1127.796,262.191,-71.233,-178.387,10.043,149.562
C08036=1127.791,262.440,-71.262,-178.383,10.046,149.562
C08037=1127.787,262.687,-71.290,-178.379,10.050,149.562
C08038=1127.783,262.935,-71.320,-178.376,10.052,149.562
C08039=1127.778,263.184,-71.349,-178.372,10.056,149.562
C08040=1127.774,263.433,-71.378,-178.368,10.059,149.561
C08041=1127.770,263.681,-71.407,-178.364,10.062,149.561
C08042=1127.766,263.930,-71.436,-178.361,10.065,149.561
C08043=1127.761,264.177,-71.465,-178.358,10.068,149.561
C08044=1127.757,264.425,-71.494,-178.354,10.071,149.560
C08045=1127.753,264.673,-71.524,-178.351,10.074,149.560
C08046=1127.749,264.922,-71.553,-178.348,10.076,149.560
C08047=1127.744,265.171,-71.582,-178.346,10.078,149.560
C08048=1127.740,265.419,-71.611,-178.343,10.081,149.560
C08049=1127.736,265.666,-71.640,-178.341,10.083,149.560
C08050=1127.731,265.915,-71.670,-178.338,10.086,149.560
C08051=1127.727,266.163,-71.699,-178.336,10.088,149.560
C08052=1127.724,266.376,-71.724,-178.334,10.090,149.560
C08053=1127.720,266.590,-71.750,-178.331,10.092,149.559
C08054=1127.716,266.804,-71.774,-178.329,10.094,149.559
C08055=1127.713,267.018,-71.800,-178.327,10.096,149.559
C08056=1127.709,267.232,-71.825,-178.325,10.098,149.559
C08057=1127.705,267.445,-71.851,-178.322,10.100,149.559
C08058=1127.702,267.659,-71.876,-178.320,10.102,149.559
C08059=1127.698,267.872,-71.901,-178.318,10.104,149.559
C08060=1127.694,268.120,-71.930,-178.315,10.107,149.559
C08061=1127.690,268.369,-71.960,-178.312,10.110,149.559
C08062=1127.686,268.617,-71.989,-178.310,10.112,149.559
C08063=1127.681,268.865,-72.019,-178.307,10.115,149.559
C08064=1127.677,269.113,-72.048,-178.304,10.117,149.559
C08065=1127.672,269.361,-72.077,-178.302,10.119,149.558
C08066=1127.668,269.609,-72.107,-178.299,10.122,149.558
C08067=1127.664,269.857,-72.136,-178.296,10.125,149.558
C08068=1127.660,270.106,-72.166,-178.294,10.127,149.558
C08069=1127.655,270.354,-72.196,-178.291,10.130,149.558
C08070=1127.651,270.603,-72.225,-178.288,10.132,149.558
C08071=1127.647,270.851,-72.255,-178.285,10.135,149.558
C08072=1127.643,271.098,-72.285,-178.283,10.137,149.558
C08073=1127.639,271.347,-72.314,-178.280,10.140,149.558
C08074=1127.634,271.595,-72.344,-178.277,10.143,149.557
C08075=1127.630,271.843,-72.373,-178.274,10.145,149.557
C08076=1127.626,272.092,-72.403,-178.271,10.148,149.557
C08077=1127.622,272.340,-72.432,-178.267,10.151,149.557
C08078=1127.617,272.588,-72.462,-178.265,10.153,149.557
C08079=1127.613,272.836,-72.492,-178.262,10.156,149.557
C08080=1127.609,273.084,-72.522,-178.259,10.159,149.557
C08081=1127.605,273.333,-72.551,-178.256,10.161,149.557
C08082=1127.601,273.581,-72.581,-178.253,10.164,149.556
C08083=1127.597,273.829,-72.611,-178.250,10.166,149.556
C08084=1127.592,274.077,-72.641,-178.247,10.169,149.556
C08085=1127.588,274.325,-72.670,-178.244,10.172,149.556
C08086=1127.584,274.573,-72.700,-178.241,10.174,149.556
C08087=1127.580,274.821,-72.730,-178.238,10.178,149.556
C08088=1127.576,275.070,-72.760,-178.235,10.181,149.556
C08089=1127.571,275.318,-72.790,-178.231,10.183,149.555
C08090=1127.567,275.566,-72.820,-178.228,10.186,149.555
C08091=1127.563,275.815,-72.849,-178.226,10.189,149.555
C08092=1127.559,276.062,-72.880,-178.222,10.191,149.555
C08093=1127.554,276.311,-72.910,-178.219,10.194,149.555
C08094=1127.550,276.559,-72.940,-178.216,10.196,149.555
C08095=1127.546,276.807,-72.969,-178.213,10.199,149.554
C08096=1127.541,277.055,-72.999,-178.209,10.202,149.554
C08097=1127.537,277.303,-73.029,-178.206,10.205,149.554
C08098=1127.533,277.551,-73.059,-178.203,10.208,149.554
C08099=1127.529,277.800,-73.090,-178.200,10.210,149.554
C08100=1127.525,278.048,-73.119,-178.196,10.214,149.554
C08101=1127.521,278.296,-73.150,-178.193,10.216,149.554
C08102=1127.516,278.544,-73.180,-178.190,10.219,149.553
C08103=1127.512,278.792,-73.210,-178.187,10.222,149.553
C08104=1127.508,279.040,-73.240,-178.183,10.225,149.553
C08105=1127.504,279.289,-73.270,-178.180,10.227,149.553
C08106=1127.500,279.537,-73.301,-178.177,10.230,149.552
C08107=1127.495,279.785,-73.331,-178.173,10.233,149.552
C08108=1127.492,279.998,-73.357,-178.170,10.235,149.552
C08109=1127.488,280.211,-73.383,-178.167,10.238,149.552
C08110=1127.485,280.425,-73.409,-178.164,10.240,149.552
C08111=1127.481,280.638,-73.435,-178.161,10.243,149.552
C08112=1127.477,280.852,-73.460,-178.158,10.245,149.551
C08113=1127.474,281.066,-73.487,-178.156,10.247,149.551
C08114=1127.470,281.279,-73.513,-178.152,10.250,149.551
C08115=1127.467,281.492,-73.539,-178.149,10.253,149.551
C08116=1127.463,281.741,-73.570,-178.146,10.255,149.551
C08117=1127.459,281.989,-73.600,-178.143,10.258,149.550
C08118=1127.454,282.237,-73.630,-178.140,10.260,149.550
C08119=1127.450,282.485,-73.660,-178.137,10.262,149.550
C08120=1127.446,282.733,-73.691,-178.134,10.265,149.550
C08121=1127.442,282.981,-73.722,-178.131,10.267,149.550
C08122=1127.437,283.229,-73.752,-178.128,10.270,149.550
C08123=1127.433,283.477,-73.782,-178.125,10.272,149.549
C08124=1127.429,283.726,-73.813,-178.122,10.275,149.549
C08125=1127.425,283.974,-73.844,-178.118,10.278,149.549
C08126=1127.421,284.222,-73.874,-178.116,10.280,149.549
C08127=1127.416,284.470,-73.905,-178.113,10.283,149.549
C08128=1127.413,284.718,-73.935,-178.109,10.286,149.548
C08129=1127.408,284.966,-73.966,-178.107,10.288,149.548
C08130=1127.404,285.214,-73.997,-178.104,10.290,149.548
C08131=1127.400,285.461,-74.027,-178.101,10.293,149.548
C08132=1127.396,285.710,-74.058,-178.097,10.295,149.548
C08133=1127.392,285.958,-74.088,-178.094,10.298,149.548
C08134=1127.387,286.206,-74.119,-178.091,10.301,149.547
C08135=1127.383,286.454,-74.150,-178.088,10.303,149.547
C08136=1127.379,286.702,-74.180,-178.085,10.306,149.547
C08137=1127.375,286.950,-74.211,-178.082,10.308,149.547
C08138=1127.371,287.199,-74.242,-178.079,10.311,149.547
C08139=1127.366,287.447,-74.273,-178.076,10.313,149.546
C08140=1127.362,287.694,-74.303,-178.073,10.315,149.546
C08141=1127.358,287.943,-74.334,-178.070,10.318,149.546
C08142=1127.354,288.191,-74.365,-178.067,10.321,149.546
C08143=1127.350,288.439,-74.396,-178.064,10.323,149.546
C08144=1127.346,288.687,-74.426,-178.061,10.326,149.546
C08145=1127.341,288.935,-74.457,-178.058,10.329,149.546
C08146=1127.337,289.183,-74.489,-178.054,10.331,149.545
C08147=1127.333,289.431,-74.519,-178.052,10.334,149.545
C08148=1127.329,289.679,-74.550,-178.048,10.336,149.545
C08149=1127.325,289.927,-74.581,-178.045,10.339,149.545
C08150=1127.320,290.175,-74.612,-178.043,10.341,149.544
C08151=1127.317,290.423,-74.644,-178.040,10.343,149.544
C08152=1127.313,290.671,-74.674,-178.036,10.346,149.544
C08153=1127.308,290.919,-74.705,-178.033,10.349,149.544
C08154=1127.304,291.168,-74.736,-178.030,10.351,149.544
C08155=1127.300,291.415,-74.767,-178.027,10.354,149.544
C08156=1127.296,291.664,-74.798,-178.024,10.357,149.544
C08157=1127.292,291.911,-74.828,-178.021,10.359,149.543
C08158=1127.288,292.159,-74.860,-178.018,10.362,149.543
C08159=1127.283,292.407,-74.891,-178.014,10.364,149.543
C08160=1127.279,292.656,-74.922,-178.012,10.367,149.543
C08161=1127.275,292.903,-74.954,-178.009,10.369,149.543
C08162=1127.271,293.152,-74.985,-178.006,10.371,149.542
C08163=1127.267,293.400,-75.016,-178.003,10.374,149.542
C08164=1127.263,293.613,-75.043,-178.000,10.376,149.542
C08165=1127.259,293.826,-75.070,-177.997,10.378,149.542
C08166=1127.256,294.040,-75.096,-177.995,10.380,149.542
C08167=1127.252,294.253,-75.123,-177.992,10.383,149.542
C08168=1127.250,294.466,-75.150,-177.989,10.385,149.542
C08169=1127.246,294.679,-75.176,-177.987,10.387,149.541
C08170=1127.242,294.893,-75.203,-177.984,10.389,149.541
C08171=1127.239,295.105,-75.230,-177.981,10.391,149.541
C08172=1127.235,295.354,-75.262,-177.979,10.394,149.541
C08173=1127.231,295.602,-75.293,-177.975,10.396,149.541
C08174=1127.226,295.850,-75.324,-177.972,10.399,149.541
C08175=1127.223,296.098,-75.356,-177.969,10.402,149.540
C08176=1127.218,296.346,-75.387,-177.966,10.404,149.540
C08177=1127.214,296.594,-75.419,-177.963,10.407,149.540
C08178=1127.210,296.842,-75.449,-177.960,10.410,149.540
C08179=1127.206,297.090,-75.481,-177.956,10.412,149.540
C08180=1127.202,297.337,-75.513,-177.954,10.414,149.539
C08181=1127.197,297.586,-75.544,-177.951,10.416,149.539
C08182=1127.193,297.834,-75.576,-177.948,10.419,149.539
C08183=1127.189,298.082,-75.608,-177.944,10.422,149.539
C08184=1127.185,298.331,-75.639,-177.942,10.424,149.539
C08185=1127.181,298.578,-75.670,-177.938,10.427,149.538
C08186=1127.177,298.826,-75.702,-177.935,10.430,149.538
C08187=1127.172,299.074,-75.733,-177.932,10.432,149.538
C08188=1127.169,299.322,-75.765,-177.929,10.435,149.538
C08189=1127.165,299.570,-75.797,-177.926,10.437,149.538
C08190=1127.161,299.817,-75.828,-177.923,10.440,149.538
C08191=1127.156,300.066,-75.860,-177.919,10.442,149.537
C08192=1127.151,300.314,-75.891,-177.916,10.445,149.537
C08193=1127.148,300.562,-75.923,-177.914,10.447,149.537
C08194=1127.144,300.810,-75.955,-177.911,10.450,149.537
C08195=1127.140,301.057,-75.987,-177.907,10.452,149.537
C08196=1127.135,301.306,-76.018,-177.905,10.455,149.537
C08197=1127.131,301.554,-76.050,-177.901,10.457,149.536
C08198=1127.127,301.801,-76.082,-177.898,10.460,149.536
C08199=1127.123,302.049,-76.113,-177.895,10.462,149.536
C08200=1127.120,302.297,-76.145,-177.892,10.465,149.536
C08201=1127.115,302.545,-76.177,-177.889,10.468,149.536
C08202=1127.111,302.793,-76.209,-177.885,10.470,149.535
C08203=1127.107,303.041,-76.241,-177.882,10.473,149.535
C08204=1127.103,303.288,-76.273,-177.879,10.475,149.535
C08205=1127.098,303.537,-76.305,-177.876,10.478,149.535
C08206=1127.095,303.785,-76.337,-177.873,10.480,149.535
C08207=1127.090,304.032,-76.368,-177.871,10.482,149.535
C08208=1127.086,304.281,-76.401,-177.867,10.485,149.534
C08209=1127.082,304.529,-76.433,-177.864,10.488,149.534
C08210=1127.078,304.776,-76.464,-177.861,10.490,149.534
C08211=1127.073,305.024,-76.497,-177.858,10.493,149.534
C08212=1127.070,305.272,-76.528,-177.855,10.495,149.534
C08213=1127.066,305.520,-76.560,-177.851,10.498,149.533
C08214=1127.061,305.768,-76.592,-177.848,10.500,149.533
C08215=1127.057,306.016,-76.624,-177.845,10.503,149.533
C08216=1127.054,306.264,-76.656,-177.842,10.506,149.533
C08217=1127.049,306.512,-76.688,-177.839,10.508,149.533
C08218=1127.045,306.760,-76.720,-177.836,10.511,149.533
C08219=1127.041,307.007,-76.753,-177.833,10.513,149.532
C08220=1127.038,307.221,-76.781,-177.830,10.515,149.532
C08221=1127.034,307.434,-76.807,-177.828,10.517,149.532
C08222=1127.030,307.647,-76.835,-177.825,10.520,149.532
C08223=1127.027,307.860,-76.863,-177.822,10.522,149.532
C08224=1127.024,308.074,-76.890,-177.820,10.523,149.532
C08225=1127.020,308.287,-76.919,-177.817,10.526,149.531
C08226=1127.016,308.500,-76.946,-177.814,10.528,149.531
C08227=1127.012,308.713,-76.974,-177.811,10.531,149.531
C08228=1127.009,308.961,-77.007,-177.809,10.533,149.531
C08229=1127.005,309.209,-77.038,-177.805,10.535,149.531
C08230=1127.001,309.457,-77.071,-177.803,10.538,149.531
C08231=1126.996,309.704,-77.102,-177.799,10.540,149.530
C08232=1126.992,309.952,-77.135,-177.796,10.543,149.530
C08233=1126.989,310.200,-77.167,-177.793,10.545,149.530
C08234=1126.984,310.448,-77.200,-177.790,10.548,149.530
C08235=1126.980,310.696,-77.233,-177.787,10.551,149.530
C08236=1126.976,310.944,-77.265,-177.783,10.553,149.529
C08237=1126.972,311.191,-77.298,-177.780,10.556,149.529
C08238=1126.968,311.439,-77.329,-177.777,10.558,149.529
C08239=1126.964,311.687,-77.363,-177.774,10.561,149.529
C08240=1126.960,311.935,-77.394,-177.771,10.564,149.529
C08241=1126.956,312.183,-77.427,-177.767,10.566,149.529
C08242=1126.952,312.431,-77.459,-177.765,10.568,149.528
C08243=1126.948,312.679,-77.492,-177.762,10.570,149.528
C08244=1126.944,312.927,-77.525,-177.759,10.573,149.528
C08245=1126.940,313.175,-77.557,-177.756,10.576,149.528
C08246=1126.935,313.422,-77.590,-177.752,10.578,149.528
C08247=1126.931,313.670,-77.623,-177.749,10.581,149.528
C08248=1126.927,313.918,-77.655,-177.746,10.583,149.527
C08249=1126.923,314.165,-77.688,-177.743,10.586,149.527
C08250=1126.919,314.413,-77.720,-177.740,10.588,149.527
C08251=1126.915,314.661,-77.753,-177.736,10.591,149.527
C08252=1126.911,314.910,-77.785,-177.734,10.594,149.527
C08253=1126.907,315.157,-77.818,-177.730,10.596,149.526
C08254=1126.903,315.405,-77.851,-177.727,10.599,149.526
C08255=1126.899,315.653,-77.883,-177.724,10.601,149.526
C08256=1126.895,315.901,-77.917,-177.721,10.604,149.526
C08257=1126.891,316.148,-77.949,-177.718,10.607,149.526
C08258=1126.887,316.396,-77.982,-177.715,10.608,149.525
C08259=1126.883,316.644,-78.015,-177.712,10.611,149.525
C08260=1126.879,316.892,-78.047,-177.709,10.613,149.525
C08261=1126.875,317.139,-78.080,-177.705,10.616,149.525
C08262=1126.871,317.388,-78.113,-177.702,10.619,149.525
C08263=1126.867,317.636,-78.146,-177.699,10.621,149.525
C08264=1126.863,317.883,-78.179,-177.696,10.623,149.524
C08265=1126.859,318.131,-78.212,-177.693,10.626,149.524
C08266=1126.855,318.378,-78.245,-177.690,10.629,149.524
C08267=1126.851,318.626,-78.278,-177.687,10.631,149.524
C08268=1126.846,318.874,-78.310,-177.683,10.634,149.524
C08269=1126.843,319.122,-78.343,-177.680,10.636,149.523
C08270=1126.839,319.370,-78.376,-177.677,10.639,149.523
C08271=1126.835,319.617,-78.409,-177.674,10.642,149.523
C08272=1126.831,319.865,-78.442,-177.670,10.644,149.523
C08273=1126.826,320.113,-78.476,-177.667,10.647,149.523
C08274=1126.822,320.361,-78.509,-177.665,10.648,149.522
C08275=1126.819,320.608,-78.541,-177.661,10.651,149.522
C08276=1126.815,320.821,-78.570,-177.659,10.654,149.522
C08277=1126.812,321.034,-78.598,-177.656,10.656,149.522
C08278=1126.808,321.247,-78.627,-177.653,10.658,149.522
C08279=1126.805,321.460,-78.655,-177.651,10.660,149.522
C08280=1126.801,321.673,-78.684,-177.648,10.662,149.521
C08281=1126.798,321.886,-78.713,-177.645,10.665,149.521
C08282=1126.794,322.100,-78.741,-177.642,10.666,149.521
C08283=1126.791,322.312,-78.769,-177.639,10.669,149.521
C08284=1126.787,322.560,-78.802,-177.637,10.671,149.521
C08285=1126.784,322.808,-78.836,-177.634,10.673,149.521
C08286=1126.779,323.056,-78.869,-177.630,10.676,149.520
C08287=1126.775,323.304,-78.902,-177.627,10.678,149.520
C08288=1126.771,323.552,-78.935,-177.624,10.681,149.520
C08289=1126.767,323.799,-78.969,-177.621,10.684,149.520
C08290=1126.763,324.046,-79.002,-177.618,10.686,149.520
C08291=1126.759,324.294,-79.035,-177.615,10.689,149.520
C08292=1126.756,324.543,-79.069,-177.611,10.691,149.519
C08293=1126.751,324.790,-79.102,-177.608,10.694,149.519
C08294=1126.747,325.038,-79.135,-177.605,10.696,149.519
C08295=1126.743,325.285,-79.169,-177.602,10.699,149.519
C08296=1126.739,325.533,-79.202,-177.598,10.701,149.518
C08297=1126.735,325.781,-79.235,-177.595,10.704,149.518
C08298=1126.732,326.029,-79.269,-177.592,10.707,149.518
C08299=1126.728,326.276,-79.303,-177.589,10.709,149.518
C08300=1126.723,326.524,-79.337,-177.586,10.712,149.518
C08301=1126.719,326.772,-79.370,-177.583,10.714,149.518
C08302=1126.715,327.019,-79.404,-177.580,10.716,149.517
C08303=1126.711,327.267,-79.437,-177.577,10.718,149.517
C08304=1126.707,327.515,-79.470,-177.574,10.721,149.517
C08305=1126.703,327.762,-79.504,-177.570,10.724,149.517
C08306=1126.699,328.010,-79.537,-177.567,10.726,149.517
C08307=1126.695,328.258,-79.570,-177.564,10.729,149.516
C08308=1126.691,328.506,-79.605,-177.561,10.731,149.516
C08309=1126.687,328.754,-79.638,-177.557,10.734,149.516
C08310=1126.683,329.001,-79.672,-177.555,10.736,149.516
C08311=1126.679,329.248,-79.705,-177.551,10.739,149.516
C08312=1126.676,329.497,-79.739,-177.548,10.741,149.515
C08313=1126.671,329.744,-79.773,-177.545,10.744,149.515
C08314=1126.667,329.992,-79.807,-177.542,10.747,149.515
C08315=1126.663,330.239,-79.841,-177.538,10.749,149.515
C08316=1126.659,330.488,-79.874,-177.535,10.751,149.515
C08317=1126.656,330.735,-79.908,-177.532,10.754,149.515
C08318=1126.651,330.982,-79.942,-177.529,10.757,149.514
C08319=1126.647,331.231,-79.976,-177.525,10.759,149.514
C08320=1126.644,331.478,-80.010,-177.523,10.761,149.514
C08321=1126.639,331.726,-80.044,-177.520,10.764,149.514
C08322=1126.636,331.973,-80.078,-177.516,10.766,149.514
C08323=1126.631,332.221,-80.111,-177.513,10.768,149.513
C08324=1126.628,332.468,-80.145,-177.510,10.771,149.513
C08325=1126.624,332.716,-80.180,-177.507,10.774,149.513
C08326=1126.619,332.964,-80.213,-177.504,10.776,149.513
C08327=1126.616,333.211,-80.247,-177.500,10.779,149.512
C08328=1126.612,333.459,-80.281,-177.497,10.781,149.512
C08329=1126.608,333.707,-80.315,-177.494,10.784,149.512
C08330=1126.604,333.954,-80.349,-177.491,10.786,149.512
C08331=1126.600,334.202,-80.383,-177.487,10.789,149.512
C08332=1126.596,334.415,-80.412,-177.485,10.791,149.512
C08333=1126.593,334.628,-80.442,-177.482,10.793,149.511
C08334=1126.589,334.840,-80.471,-177.480,10.795,149.511
C08335=1126.586,335.053,-80.500,-177.476,10.798,149.511
C08336=1126.583,335.266,-80.530,-177.474,10.800,149.511
C08337=1126.579,335.479,-80.559,-177.471,10.801,149.511
C08338=1126.576,335.692,-80.588,-177.468,10.804,149.511
C08339=1126.572,335.905,-80.618,-177.466,10.806,149.510
C08340=1126.569,336.152,-80.652,-177.462,10.808,149.510
C08341=1126.564,336.400,-80.686,-177.459,10.811,149.510
C08342=1126.561,336.648,-80.720,-177.456,10.813,149.510
C08343=1126.556,336.896,-80.754,-177.453,10.816,149.510
C08344=1126.553,337.143,-80.788,-177.449,10.818,149.509
C08345=1126.549,337.391,-80.823,-177.446,10.821,149.509
C08346=1126.545,337.638,-80.857,-177.443,10.824,149.509
C08347=1126.541,337.886,-80.892,-177.440,10.826,149.509
C08348=1126.537,338.133,-80.925,-177.437,10.829,149.509
C08349=1126.533,338.381,-80.960,-177.433,10.831,149.508
C08350=1126.529,338.628,-80.994,-177.430,10.834,149.508
C08351=1126.525,338.877,-81.029,-177.427,10.836,149.508
C08352=1126.521,339.124,-81.063,-177.424,10.838,149.508
C08353=1126.517,339.371,-81.097,-177.421,10.840,149.508
C08354=1126.514,339.619,-81.132,-177.418,10.843,149.507
C08355=1126.509,339.866,-81.166,-177.415,10.846,149.507
C08356=1126.505,340.114,-81.201,-177.411,10.848,149.507
C08357=1126.501,340.362,-81.235,-177.408,10.850,149.507
C08358=1126.497,340.610,-81.270,-177.405,10.853,149.507
C08359=1126.493,340.857,-81.303,-177.401,10.855,149.506
C08360=1126.489,341.105,-81.338,-177.399,10.858,149.506
C08361=1126.485,341.352,-81.373,-177.395,10.861,149.506
C08362=1126.482,341.600,-81.408,-177.392,10.863,149.506
C08363=1126.477,341.847,-81.442,-177.389,10.866,149.506
C08364=1126.473,342.095,-81.477,-177.385,10.868,149.505
C08365=1126.470,342.342,-81.511,-177.382,10.871,149.505
C08366=1126.466,342.590,-81.546,-177.379,10.873,149.505
C08367=1126.462,342.838,-81.581,-177.376,10.876,149.505
C08368=1126.458,343.085,-81.615,-177.372,10.878,149.505
C08369=1126.454,343.333,-81.650,-177.369,10.881,149.504
C08370=1126.450,343.580,-81.685,-177.366,10.883,149.504
C08371=1126.446,343.828,-81.720,-177.363,10.886,149.504
C08372=1126.442,344.075,-81.754,-177.360,10.888,149.504
C08373=1126.438,344.323,-81.789,-177.357,10.890,149.504
C08374=1126.434,344.570,-81.824,-177.354,10.892,149.503
C08375=1126.430,344.818,-81.859,-177.350,10.895,149.503
C08376=1126.427,345.066,-81.893,-177.347,10.897,149.503
C08377=1126.422,345.313,-81.928,-177.344,10.900,149.503
C08378=1126.418,345.561,-81.963,-177.341,10.903,149.503
C08379=1126.414,345.808,-81.998,-177.337,10.905,149.502
C08380=1126.411,346.055,-82.032,-177.334,10.908,149.502
C08381=1126.407,346.304,-82.067,-177.331,10.910,149.502
C08382=1126.403,346.550,-82.102,-177.327,10.912,149.502
C08383=1126.399,346.798,-82.137,-177.324,10.915,149.502
C08384=1126.395,347.046,-82.173,-177.321,10.918,149.501
C08385=1126.391,347.293,-82.207,-177.318,10.920,149.501
C08386=1126.388,347.541,-82.242,-177.315,10.923,149.501
C08387=1126.383,347.788,-82.277,-177.311,10.925,149.501
C08388=1126.380,348.001,-82.307,-177.309,10.927,149.501
C08389=1126.376,348.214,-82.337,-177.306,10.930,149.500
C08390=1126.373,348.427,-82.367,-177.303,10.931,149.500
C08391=1126.370,348.639,-82.397,-177.300,10.933,149.500
C08392=1126.367,348.852,-82.428,-177.297,10.936,149.500
C08393=1126.363,349.064,-82.458,-177.295,10.937,149.500
C08394=1126.360,349.277,-82.488,-177.292,10.940,149.500
C08395=1126.356,349.490,-82.519,-177.289,10.942,149.499
C08396=1126.352,349.738,-82.553,-177.286,10.944,149.499
C08397=1126.348,349.985,-82.589,-177.282,10.948,149.499
C08398=1126.344,350.232,-82.624,-177.278,10.950,149.498
C08399=1126.340,350.480,-82.659,-177.275,10.952,149.498
C08400=1126.338,350.728,-82.694,-177.271,10.955,149.498
C08401=1126.333,350.974,-82.729,-177.268,10.958,149.498
C08402=1126.330,351.222,-82.765,-177.264,10.960,149.498
C08403=1126.326,351.470,-82.800,-177.260,10.963,149.497
C08404=1126.322,351.717,-82.835,-177.257,10.966,149.497
C08405=1126.318,351.964,-82.870,-177.253,10.968,149.497
C08406=1126.314,352.212,-82.906,-177.250,10.971,149.497
C08407=1126.310,352.460,-82.941,-177.246,10.974,149.496
C08408=1126.306,352.707,-82.976,-177.242,10.976,149.496
C08409=1126.301,352.955,-83.012,-177.239,10.978,149.496
C08410=1126.298,353.202,-83.047,-177.236,10.981,149.496
C08411=1126.294,353.450,-83.083,-177.232,10.984,149.495
C08412=1126.290,353.697,-83.119,-177.228,10.986,149.495
C08413=1126.287,353.945,-83.154,-177.225,10.989,149.495
C08414=1126.283,354.191,-83.189,-177.222,10.991,149.494
C08415=1126.279,354.439,-83.225,-177.218,10.994,149.494
C08416=1126.275,354.686,-83.260,-177.214,10.997,149.494
C08417=1126.271,354.934,-83.295,-177.211,10.999,149.494
C08418=1126.268,355.182,-83.331,-177.207,11.001,149.493
C08419=1126.264,355.429,-83.366,-177.204,11.004,149.493
C08420=1126.259,355.676,-83.403,-177.200,11.006,149.493
C08421=1126.256,355.923,-83.438,-177.196,11.009,149.493
C08422=1126.252,356.171,-83.474,-177.193,11.012,149.492
C08423=1126.248,356.418,-83.509,-177.190,11.014,149.492
C08424=1126.245,356.666,-83.545,-177.186,11.016,149.492
C08425=1126.241,356.913,-83.581,-177.183,11.019,149.492
C08426=1126.236,357.161,-83.617,-177.179,11.021,149.491
C08427=1126.233,357.409,-83.652,-177.176,11.024,149.491
C08428=1126.229,357.656,-83.687,-177.172,11.026,149.491
C08429=1126.225,357.903,-83.723,-177.168,11.029,149.491
C08430=1126.222,358.150,-83.759,-177.165,11.032,149.490
C08431=1126.217,358.398,-83.795,-177.162,11.034,149.490
C08432=1126.213,358.645,-83.831,-177.158,11.036,149.490
C08433=1126.210,358.893,-83.866,-177.155,11.039,149.489
C08434=1126.206,359.140,-83.902,-177.151,11.041,149.489
C08435=1126.202,359.387,-83.939,-177.148,11.044,149.489
C08436=1126.198,359.635,-83.974,-177.144,11.046,149.489
C08437=1126.195,359.882,-84.010,-177.141,11.048,149.488
C08438=1126.191,360.130,-84.047,-177.138,11.051,149.488
C08439=1126.187,360.377,-84.082,-177.135,11.053,149.488
C08440=1126.183,360.625,-84.118,-177.131,11.055,149.488
C08441=1126.180,360.872,-84.154,-177.128,11.058,149.487
C08442=1126.176,361.119,-84.190,-177.124,11.060,149.487
C08443=1126.172,361.367,-84.226,-177.121,11.063,149.487
C08444=1126.168,361.579,-84.257,-177.118,11.065,149.487
C08445=1126.165,361.791,-84.288,-177.115,11.067,149.486
C08446=1126.162,362.004,-84.319,-177.112,11.069,149.486
C08447=1126.158,362.217,-84.350,-177.109,11.071,149.486
C08448=1126.155,362.429,-84.381,-177.106,11.073,149.486
C08449=1126.152,362.642,-84.412,-177.103,11.075,149.486
C08450=1126.148,362.854,-84.443,-177.100,11.077,149.485
C08451=1126.145,363.067,-84.474,-177.098,11.079,149.485
C08452=1126.142,363.314,-84.510,-177.094,11.081,149.485
C08453=1126.138,363.561,-84.547,-177.091,11.084,149.485
C08454=1126.134,363.809,-84.582,-177.088,11.086,149.484
C08455=1126.130,364.056,-84.619,-177.084,11.088,149.484
C08456=1126.126,364.303,-84.655,-177.081,11.091,149.484
C08457=1126.123,364.550,-84.691,-177.077,11.093,149.484
C08458=1126.119,364.799,-84.727,-177.074,11.096,149.483
C08459=1126.116,365.046,-84.764,-177.071,11.098,149.483
C08460=1126.112,365.293,-84.801,-177.068,11.100,149.483
C08461=1126.108,365.540,-84.836,-177.064,11.103,149.483
C08462=1126.104,365.788,-84.873,-177.061,11.105,149.482
C08463=1126.100,366.035,-84.909,-177.058,11.107,149.482
C08464=1126.096,366.282,-84.945,-177.055,11.109,149.482
C08465=1126.092,366.529,-84.982,-177.051,11.112,149.482
C08466=1126.088,366.777,-85.018,-177.048,11.114,149.481
C08467=1126.084,367.024,-85.055,-177.045,11.117,149.481
C08468=1126.081,367.271,-85.091,-177.041,11.119,149.481
C08469=1126.077,367.518,-85.128,-177.038,11.122,149.481
C08470=1126.073,367.766,-85.163,-177.035,11.124,149.481
C08471=1126.070,368.014,-85.201,-177.032,11.126,149.480
C08472=1126.066,368.261,-85.237,-177.029,11.128,149.480
C08473=1126.062,368.508,-85.274,-177.025,11.131,149.480
C08474=1126.058,368.755,-85.310,-177.022,11.133,149.480
C08475=1126.054,369.002,-85.346,-177.019,11.136,149.479
C08476=1126.050,369.250,-85.383,-177.016,11.138,149.479
C08477=1126.046,369.497,-85.420,-177.013,11.140,149.479
C08478=1126.043,369.744,-85.456,-177.010,11.142,149.479
C08479=1126.039,369.992,-85.493,-177.006,11.145,149.479
C08480=1126.035,370.239,-85.530,-177.003,11.147,149.478
C08481=1126.032,370.486,-85.566,-177.000,11.150,149.478
C08482=1126.028,370.733,-85.603,-176.997,11.151,149.478
C08483=1126.023,370.981,-85.639,-176.994,11.154,149.478
C08484=1126.021,371.228,-85.676,-176.990,11.156,149.478
C08485=1126.017,371.475,-85.713,-176.987,11.159,149.477
C08486=1126.013,371.723,-85.750,-176.984,11.161,149.477
C08487=1126.008,371.970,-85.787,-176.981,11.163,149.477
C08488=1126.005,372.217,-85.823,-176.978,11.166,149.477
C08489=1126.002,372.465,-85.860,-176.975,11.168,149.476
C08490=1125.997,372.712,-85.897,-176.971,11.171,149.476
C08491=1125.993,372.959,-85.934,-176.969,11.172,149.476
C08492=1125.990,373.206,-85.970,-176.965,11.175,149.476
C08493=1125.987,373.454,-86.007,-176.962,11.178,149.476
C08494=1125.983,373.700,-86.045,-176.959,11.180,149.476
C08495=1125.979,373.947,-86.082,-176.956,11.182,149.475
C08496=1125.975,374.194,-86.118,-176.953,11.184,149.475
C08497=1125.972,374.442,-86.155,-176.950,11.187,149.475
C08498=1125.968,374.689,-86.192,-176.947,11.189,149.475
C08499=1125.964,374.937,-86.229,-176.944,11.191,149.475
C08500=1125.961,375.149,-86.261,-176.941,11.194,149.474
C08501=1125.957,375.362,-86.293,-176.939,11.196,149.474
C08502=1125.954,375.574,-86.325,-176.936,11.197,149.474
C08503=1125.951,375.786,-86.356,-176.934,11.199,149.474
C08504=1125.948,375.999,-86.389,-176.931,11.201,149.474
C08505=1125.945,376.211,-86.420,-176.928,11.204,149.474
C08506=1125.941,376.423,-86.452,-176.925,11.206,149.474
C08507=1125.938,376.636,-86.483,-176.923,11.208,149.474
C08508=1125.934,376.883,-86.521,-176.920,11.210,149.473
C08509=1125.930,377.130,-86.558,-176.918,11.212,149.473
C08510=1125.926,377.377,-86.595,-176.914,11.215,149.473
C08511=1125.923,377.625,-86.632,-176.911,11.217,149.473
C08512=1125.920,377.871,-86.669,-176.909,11.219,149.473
C08513=1125.916,378.119,-86.706,-176.905,11.222,149.473
C08514=1125.912,378.366,-86.743,-176.903,11.224,149.473
C08515=1125.908,378.613,-86.781,-176.899,11.227,149.472
C08516=1125.904,378.860,-86.818,-176.897,11.229,149.472
C08517=1125.901,379.108,-86.855,-176.894,11.231,149.472
C08518=1125.897,379.355,-86.893,-176.890,11.234,149.472
C08519=1125.893,379.602,-86.929,-176.888,11.236,149.472
C08520=1125.890,379.849,-86.967,-176.885,11.238,149.472
C08521=1125.886,380.096,-87.004,-176.882,11.241,149.472
C08522=1125.882,380.343,-87.041,-176.880,11.243,149.472
C08523=1125.878,380.591,-87.079,-176.876,11.246,149.471
C08524=1125.874,380.838,-87.116,-176.873,11.249,149.471
C08525=1125.871,381.085,-87.154,-176.871,11.250,149.471
C08526=1125.867,381.332,-87.191,-176.868,11.253,149.471
C08527=1125.863,381.579,-87.228,-176.865,11.256,149.471
C08528=1125.860,381.827,-87.265,-176.862,11.258,149.471
C08529=1125.856,382.073,-87.303,-176.859,11.260,149.471
C08530=1125.853,382.321,-87.341,-176.857,11.263,149.471
C08531=1125.848,382.568,-87.378,-176.854,11.265,149.471
C08532=1125.844,382.815,-87.416,-176.851,11.268,149.471
C08533=1125.841,383.063,-87.453,-176.848,11.271,149.471
C08534=1125.837,383.309,-87.491,-176.846,11.273,149.471
C08535=1125.834,383.557,-87.529,-176.844,11.275,149.471
C08536=1125.830,383.804,-87.566,-176.842,11.277,149.471
C08537=1125.826,384.051,-87.604,-176.840,11.278,149.471
C08538=1125.822,384.298,-87.640,-176.838,11.281,149.471
C08539=1125.818,384.545,-87.678,-176.837,11.282,149.471
C08540=1125.815,384.792,-87.716,-176.835,11.284,149.471
C08541=1125.810,385.039,-87.753,-176.834,11.286,149.471
C08542=1125.807,385.287,-87.791,-176.832,11.288,149.471
C08543=1125.803,385.533,-87.829,-176.831,11.290,149.471
C08544=1125.800,385.781,-87.867,-176.829,11.292,149.471
C08545=1125.796,386.028,-87.904,-176.828,11.294,149.471
C08546=1125.793,386.275,-87.942,-176.826,11.296,149.472
C08547=1125.789,386.522,-87.979,-176.824,11.298,149.472
C08548=1125.785,386.770,-88.017,-176.823,11.300,149.472
C08549=1125.781,387.016,-88.055,-176.821,11.303,149.472
C08550=1125.778,387.264,-88.093,-176.819,11.304,149.472
C08551=1125.774,387.510,-88.130,-176.818,11.307,149.472
C08552=1125.771,387.758,-88.168,-176.817,11.308,149.472
C08553=1125.766,388.005,-88.206,-176.815,11.311,149.473
C08554=1125.763,388.252,-88.243,-176.814,11.313,149.473
C08555=1125.759,388.499,-88.281,-176.812,11.315,149.473
C08556=1125.756,388.711,-88.314,-176.811,11.317,149.473
C08557=1125.753,388.923,-88.346,-176.810,11.318,149.473
C08558=1125.750,389.136,-88.378,-176.808,11.321,149.474
C08559=1125.746,389.348,-88.411,-176.807,11.323,149.474
C08560=1125.743,389.560,-88.443,-176.806,11.325,149.474
C08561=1125.740,389.773,-88.476,-176.805,11.326,149.474
C08562=1125.737,389.985,-88.508,-176.804,11.329,149.474
C08563=1125.734,390.197,-88.540,-176.803,11.331,149.475
C08564=1125.730,390.444,-88.578,-176.801,11.333,149.475
C08565=1125.726,390.692,-88.616,-176.800,11.335,149.475
C08566=1125.723,390.938,-88.654,-176.799,11.338,149.475
C08567=1125.720,391.185,-88.692,-176.797,11.340,149.476
C08568=1125.716,391.432,-88.729,-176.796,11.342,149.476
C08569=1125.712,391.680,-88.768,-176.795,11.345,149.476
C08570=1125.708,391.927,-88.805,-176.793,11.348,149.477
C08571=1125.705,392.174,-88.843,-176.793,11.350,149.477
C08572=1125.701,392.421,-88.881,-176.791,11.353,149.477
C08573=1125.697,392.668,-88.919,-176.790,11.355,149.478
C08574=1125.694,392.915,-88.957,-176.789,11.357,149.478
C08575=1125.690,393.162,-88.994,-176.788,11.360,149.479
C08576=1125.686,393.410,-89.033,-176.786,11.363,149.479
C08577=1125.682,393.656,-89.071,-176.785,11.366,149.479
C08578=1125.679,393.903,-89.108,-176.784,11.368,149.480
C08579=1125.675,394.151,-89.147,-176.783,11.371,149.480
C08580=1125.671,394.398,-89.185,-176.782,11.374,149.480
C08581=1125.668,394.645,-89.223,-176.781,11.377,149.481
C08582=1125.663,394.892,-89.261,-176.780,11.378,149.481
C08583=1125.660,395.139,-89.299,-176.779,11.381,149.482
C08584=1125.657,395.386,-89.336,-176.778,11.384,149.482
C08585=1125.653,395.633,-89.375,-176.777,11.387,149.483
C08586=1125.649,395.880,-89.413,-176.776,11.390,149.483
C08587=1125.646,396.127,-89.450,-176.775,11.393,149.484
C08588=1125.642,396.375,-89.489,-176.774,11.396,149.484
C08589=1125.638,396.621,-89.526,-176.773,11.399,149.485
C08590=1125.635,396.868,-89.564,-176.772,11.402,149.485
C08591=1125.631,397.115,-89.604,-176.771,11.405,149.486
C08592=1125.627,397.362,-89.641,-176.770,11.408,149.486
C08593=1125.623,397.609,-89.680,-176.769,11.411,149.487
C08594=1125.620,397.856,-89.717,-176.769,11.413,149.487
C08595=1125.616,398.103,-89.755,-176.767,11.416,149.488
C08596=1125.612,398.351,-89.794,-176.767,11.420,149.489
C08597=1125.609,398.597,-89.831,-176.766,11.423,149.489
C08598=1125.605,398.845,-89.870,-176.765,11.426,149.490
C08599=1125.601,399.091,-89.908,-176.764,11.429,149.490
C08600=1125.598,399.338,-89.946,-176.763,11.432,149.491
C08601=1125.594,399.586,-89.985,-176.762,11.436,149.492
C08602=1125.590,399.832,-90.022,-176.762,11.439,149.492
C08603=1125.586,400.080,-90.061,-176.761,11.442,149.493
C08604=1125.583,400.327,-90.099,-176.760,11.445,149.494
C08605=1125.579,400.574,-90.138,-176.759,11.449,149.494
C08606=1125.576,400.821,-90.175,-176.759,11.452,149.495
C08607=1125.572,401.068,-90.214,-176.758,11.455,149.496
C08608=1125.568,401.315,-90.252,-176.757,11.459,149.496
C08609=1125.565,401.562,-90.290,-176.757,11.462,149.497
C08610=1125.561,401.809,-90.329,-176.756,11.466,149.498
C08611=1125.558,402.056,-90.366,-176.755,11.469,149.499
C08612=1125.554,402.268,-90.399,-176.755,11.472,149.499
C08613=1125.552,402.481,-90.433,-176.755,11.475,149.500
C08614=1125.548,402.693,-90.465,-176.754,11.478,149.501
C08615=1125.545,402.905,-90.498,-176.754,11.481,149.501
C08616=1125.541,403.117,-90.531,-176.753,11.484,149.502
C08617=1125.538,403.329,-90.564,-176.753,11.488,149.503
C08618=1125.535,403.541,-90.597,-176.752,11.490,149.503
C08619=1125.533,403.753,-90.630,-176.752,11.494,149.504
C08620=1125.528,404.000,-90.668,-176.751,11.497,149.505
C08621=1125.525,404.247,-90.706,-176.751,11.501,149.506
C08622=1125.522,404.494,-90.745,-176.751,11.505,149.507
C08623=1125.518,404.741,-90.783,-176.750,11.508,149.508
C08624=1125.514,404.988,-90.821,-176.750,11.513,149.508
C08625=1125.511,405.235,-90.860,-176.749,11.516,149.509
C08626=1125.507,405.483,-90.899,-176.749,11.520,149.510
C08627=1125.503,405.729,-90.937,-176.749,11.524,149.511
C08628=1125.500,405.976,-90.976,-176.749,11.528,149.512
C08629=1125.496,406.224,-91.014,-176.748,11.532,149.513
C08630=1125.492,406.470,-91.052,-176.747,11.536,149.514
C08631=1125.488,406.717,-91.091,-176.747,11.540,149.515
C08632=1125.485,406.965,-91.129,-176.747,11.543,149.516
C08633=1125.482,407.211,-91.168,-176.747,11.548,149.517
C08634=1125.478,407.458,-91.206,-176.747,11.552,149.518
C08635=1125.474,407.705,-91.245,-176.746,11.556,149.519
C08636=1125.470,407.953,-91.283,-176.746,11.560,149.520
C08637=1125.467,408.199,-91.322,-176.746,11.565,149.521
C08638=1125.463,408.446,-91.360,-176.746,11.569,149.522
C08639=1125.460,408.693,-91.398,-176.746,11.573,149.523
C08640=1125.456,408.940,-91.437,-176.745,11.577,149.524
C08641=1125.453,409.188,-91.475,-176.746,11.581,149.525
C08642=1125.449,409.434,-91.514,-176.746,11.585,149.526
C08643=1125.445,409.681,-91.553,-176.745,11.590,149.528
C08644=1125.442,409.928,-91.591,-176.745,11.594,149.529
C08645=1125.438,410.176,-91.630,-176.745,11.599,149.530
C08646=1125.434,410.422,-91.669,-176.745,11.603,149.531
C08647=1125.431,410.669,-91.708,-176.745,11.608,149.532
C08648=1125.427,410.916,-91.746,-176.745,11.613,149.533
C08649=1125.423,411.163,-91.785,-176.746,11.617,149.535
C08650=1125.419,411.410,-91.823,-176.745,11.622,149.536
C08651=1125.416,411.657,-91.862,-176.746,11.626,149.537
C08652=1125.413,411.904,-91.900,-176.745,11.631,149.538
C08653=1125.409,412.151,-91.939,-176.746,11.635,149.540
C08654=1125.405,412.398,-91.978,-176.746,11.641,149.541
C08655=1125.402,412.644,-92.016,-176.746,11.645,149.542
C08656=1125.398,412.891,-92.055,-176.746,11.650,149.544
C08657=1125.394,413.139,-92.094,-176.746,11.655,149.545
C08658=1125.391,413.386,-92.133,-176.747,11.660,149.546
C08659=1125.388,413.633,-92.172,-176.747,11.665,149.548
C08660=1125.383,413.879,-92.210,-176.747,11.669,149.549
C08661=1125.380,414.126,-92.249,-176.747,11.675,149.550
C08662=1125.378,414.373,-92.288,-176.747,11.680,149.552
C08663=1125.375,414.620,-92.326,-176.748,11.685,149.553
C08664=1125.374,414.868,-92.365,-176.748,11.690,149.554
C08665=1125.373,415.115,-92.403,-176.749,11.695,149.556
C08666=1125.373,415.362,-92.441,-176.749,11.700,149.557
C08667=1125.373,415.609,-92.480,-176.750,11.706,149.559
C08668=1125.373,415.821,-92.512,-176.750,11.710,149.560
C08669=1125.375,416.032,-92.545,-176.750,11.714,149.561
C08670=1125.376,416.245,-92.578,-176.751,11.718,149.562
C08671=1125.378,416.456,-92.610,-176.752,11.723,149.564
C08672=1125.380,416.668,-92.643,-176.752,11.727,149.565
C08673=1125.384,416.881,-92.675,-176.753,11.732,149.566
C08674=1125.386,417.092,-92.708,-176.753,11.737,149.568
C08675=1125.389,417.305,-92.740,-176.753,11.741,149.569
C08676=1124.970,417.305,-92.803,-176.746,11.746,149.568
C08677=1124.967,417.092,-92.770,-176.745,11.741,149.567
C08678=1124.964,416.880,-92.738,-176.745,11.737,149.566
C08679=1124.961,416.668,-92.706,-176.745,11.732,149.564
C08680=1124.959,416.456,-92.673,-176.744,11.727,149.563
C08681=1124.957,416.245,-92.641,-176.744,11.723,149.562
C08682=1124.956,416.032,-92.607,-176.743,11.718,149.561
C08683=1124.954,415.820,-92.575,-176.743,11.714,149.559
C08684=1124.954,415.608,-92.542,-176.743,11.709,149.558
C08685=1124.953,415.361,-92.504,-176.742,11.704,149.557
C08686=1124.954,415.114,-92.465,-176.742,11.699,149.555
C08687=1124.954,414.867,-92.428,-176.742,11.694,149.554
C08688=1124.956,414.621,-92.388,-176.741,11.689,149.552
C08689=1124.958,414.373,-92.349,-176.741,11.684,149.551
C08690=1124.961,414.126,-92.311,-176.741,11.678,149.549
C08691=1124.964,413.879,-92.273,-176.740,11.674,149.548
C08692=1124.968,413.632,-92.233,-176.740,11.669,149.547
C08693=1124.972,413.385,-92.195,-176.740,11.664,149.545
C08694=1124.974,413.138,-92.156,-176.740,11.659,149.544
C08695=1124.979,412.892,-92.117,-176.740,11.654,149.543
C08696=1124.983,412.644,-92.079,-176.740,11.649,149.541
C08697=1124.986,412.398,-92.040,-176.739,11.644,149.540
C08698=1124.989,412.151,-92.001,-176.740,11.639,149.539
C08699=1124.993,411.903,-91.962,-176.739,11.635,149.538
C08700=1124.997,411.657,-91.924,-176.739,11.630,149.536
C08701=1125.000,411.410,-91.886,-176.739,11.626,149.535
C08702=1125.004,411.163,-91.846,-176.739,11.621,149.534
C08703=1125.007,410.916,-91.808,-176.740,11.616,149.533
C08704=1125.011,410.668,-91.769,-176.739,11.612,149.532
C08705=1125.015,410.422,-91.730,-176.740,11.607,149.530
C08706=1125.018,410.175,-91.692,-176.740,11.603,149.529
C08707=1125.022,409.928,-91.653,-176.739,11.598,149.528
C08708=1125.026,409.680,-91.615,-176.740,11.593,149.527
C08709=1125.029,409.434,-91.576,-176.740,11.589,149.526
C08710=1125.033,409.187,-91.538,-176.740,11.585,149.525
C08711=1125.036,408.940,-91.499,-176.740,11.581,149.524
C08712=1125.040,408.693,-91.461,-176.741,11.576,149.523
C08713=1125.044,408.446,-91.422,-176.741,11.572,149.522
C08714=1125.047,408.199,-91.384,-176.741,11.568,149.521
C08715=1125.051,407.952,-91.344,-176.741,11.563,149.520
C08716=1125.054,407.705,-91.307,-176.741,11.559,149.518
C08717=1125.058,407.459,-91.268,-176.742,11.555,149.518
C08718=1125.062,407.211,-91.230,-176.742,11.551,149.516
C08719=1125.065,406.964,-91.190,-176.742,11.547,149.515
C08720=1125.069,406.717,-91.152,-176.742,11.543,149.515
C08721=1125.073,406.471,-91.114,-176.743,11.538,149.513
C08722=1125.077,406.223,-91.075,-176.743,11.535,149.513
C08723=1125.080,405.976,-91.037,-176.743,11.531,149.512
C08724=1125.083,405.729,-90.998,-176.744,11.527,149.511
C08725=1125.087,405.483,-90.960,-176.744,11.523,149.510
C08726=1125.091,405.236,-90.921,-176.745,11.519,149.509
C08727=1125.094,404.988,-90.883,-176.745,11.515,149.508
C08728=1125.099,404.741,-90.845,-176.746,11.511,149.507
C08729=1125.102,404.494,-90.806,-176.746,11.507,149.506
C08730=1125.105,404.247,-90.768,-176.746,11.503,149.505
C08731=1125.109,404.000,-90.729,-176.747,11.500,149.505
C08732=1125.113,403.754,-90.691,-176.747,11.496,149.504
C08733=1125.116,403.541,-90.658,-176.748,11.493,149.503
C08734=1125.119,403.329,-90.625,-176.749,11.490,149.502
C08735=1125.122,403.117,-90.592,-176.749,11.487,149.502
C08736=1125.125,402.905,-90.559,-176.750,11.484,149.501
C08737=1125.128,402.693,-90.527,-176.750,11.481,149.500
C08738=1125.131,402.481,-90.494,-176.751,11.477,149.500
C08739=1125.135,402.269,-90.461,-176.751,11.475,149.499
C08740=1125.137,402.056,-90.427,-176.752,11.471,149.498
C08741=1125.142,401.809,-90.389,-176.752,11.468,149.498
C08742=1125.145,401.562,-90.351,-176.753,11.464,149.497
C08743=1125.149,401.315,-90.313,-176.753,11.461,149.496
C08744=1125.153,401.069,-90.274,-176.754,11.458,149.495
C08745=1125.156,400.821,-90.236,-176.755,11.454,149.495
C08746=1125.160,400.574,-90.198,-176.756,11.451,149.494
C08747=1125.163,400.327,-90.160,-176.756,11.448,149.493
C08748=1125.167,400.080,-90.122,-176.757,11.444,149.493
C08749=1125.170,399.833,-90.083,-176.758,11.441,149.492
C08750=1125.175,399.586,-90.045,-176.759,11.438,149.491
C08751=1125.178,399.339,-90.007,-176.759,11.435,149.491
C08752=1125.182,399.092,-89.969,-176.761,11.432,149.490
C08753=1125.186,398.845,-89.931,-176.761,11.428,149.489
C08754=1125.189,398.598,-89.892,-176.762,11.425,149.489
C08755=1125.193,398.351,-89.854,-176.763,11.422,149.488
C08756=1125.196,398.104,-89.816,-176.764,11.419,149.488
C08757=1125.200,397.856,-89.778,-176.765,11.416,149.487
C08758=1125.204,397.610,-89.740,-176.766,11.413,149.487
C08759=1125.207,397.362,-89.702,-176.767,11.409,149.486
C08760=1125.212,397.116,-89.664,-176.768,11.406,149.486
C08761=1125.215,396.868,-89.626,-176.769,11.403,149.485
C08762=1125.218,396.621,-89.587,-176.770,11.400,149.484
C08763=1125.222,396.375,-89.549,-176.770,11.398,149.484
C08764=1125.225,396.127,-89.511,-176.771,11.395,149.483
C08765=1125.230,395.881,-89.473,-176.773,11.392,149.483
C08766=1125.233,395.633,-89.435,-176.774,11.389,149.483
C08767=1125.236,395.386,-89.397,-176.775,11.386,149.482
C08768=1125.241,395.139,-89.359,-176.776,11.383,149.482
C08769=1125.244,394.892,-89.321,-176.777,11.380,149.481
C08770=1125.248,394.645,-89.283,-176.778,11.378,149.481
C08771=1125.252,394.398,-89.245,-176.779,11.375,149.480
C08772=1125.256,394.151,-89.207,-176.780,11.372,149.480
C08773=1125.259,393.904,-89.169,-176.782,11.370,149.479
C08774=1125.263,393.656,-89.131,-176.783,11.367,149.479
C08775=1125.266,393.410,-89.093,-176.784,11.365,149.479
C08776=1125.270,393.162,-89.055,-176.785,11.362,149.478
C08777=1125.274,392.916,-89.017,-176.786,11.359,149.478
C08778=1125.277,392.668,-88.979,-176.788,11.356,149.477
C08779=1125.281,392.422,-88.942,-176.789,11.354,149.477
C08780=1125.285,392.174,-88.903,-176.790,11.352,149.477
C08781=1125.288,391.927,-88.865,-176.792,11.349,149.477
C08782=1125.292,391.680,-88.828,-176.793,11.346,149.476
C08783=1125.296,391.432,-88.790,-176.794,11.344,149.476
C08784=1125.300,391.186,-88.752,-176.795,11.342,149.476
C08785=1125.303,390.938,-88.714,-176.797,11.339,149.475
C08786=1125.307,390.692,-88.677,-176.798,11.337,149.475
C08787=1125.310,390.444,-88.639,-176.799,11.334,149.475
C08788=1125.315,390.198,-88.601,-176.801,11.332,149.474
C08789=1125.318,389.986,-88.569,-176.802,11.330,149.474
C08790=1125.321,389.773,-88.536,-176.803,11.328,149.474
C08791=1125.324,389.560,-88.503,-176.804,11.326,149.474
C08792=1125.327,389.348,-88.471,-176.806,11.324,149.474
C08793=1125.330,389.136,-88.439,-176.806,11.322,149.473
C08794=1125.334,388.923,-88.406,-176.808,11.320,149.473
C08795=1125.336,388.711,-88.374,-176.809,11.318,149.473
C08796=1125.340,388.499,-88.341,-176.810,11.316,149.473
C08797=1125.344,388.253,-88.304,-176.812,11.314,149.473
C08798=1125.347,388.005,-88.266,-176.813,11.312,149.472
C08799=1125.351,387.759,-88.228,-176.815,11.310,149.472
C08800=1125.354,387.511,-88.190,-176.817,11.307,149.472
C08801=1125.359,387.264,-88.153,-176.818,11.305,149.472
C08802=1125.362,387.017,-88.115,-176.820,11.303,149.472
C08803=1125.366,386.770,-88.077,-176.821,11.301,149.472
C08804=1125.369,386.523,-88.039,-176.823,11.299,149.472
C08805=1125.373,386.276,-88.003,-176.825,11.297,149.471
C08806=1125.377,386.028,-87.964,-176.826,11.295,149.471
C08807=1125.381,385.781,-87.926,-176.827,11.292,149.471
C08808=1125.384,385.534,-87.889,-176.829,11.291,149.471
C08809=1125.388,385.287,-87.852,-176.831,11.289,149.471
C08810=1125.391,385.040,-87.814,-176.832,11.287,149.471
C08811=1125.395,384.793,-87.776,-176.834,11.285,149.471
C08812=1125.398,384.545,-87.739,-176.835,11.283,149.471
C08813=1125.403,384.298,-87.701,-176.837,11.281,149.471
C08814=1125.407,384.052,-87.663,-176.839,11.279,149.471
C08815=1125.410,383.804,-87.626,-176.841,11.277,149.470
C08816=1125.414,383.557,-87.588,-176.843,11.275,149.470
C08817=1125.417,383.309,-87.551,-176.845,11.273,149.470
C08818=1125.421,383.063,-87.514,-176.847,11.271,149.470
C08819=1125.424,382.816,-87.476,-176.850,11.268,149.470
C08820=1125.428,382.568,-87.439,-176.853,11.266,149.471
C08821=1125.432,382.322,-87.401,-176.856,11.264,149.471
C08822=1125.436,382.074,-87.364,-176.858,11.261,149.471
C08823=1125.440,381.827,-87.326,-176.862,11.258,149.471
C08824=1125.443,381.580,-87.288,-176.864,11.256,149.471
C08825=1125.448,381.333,-87.251,-176.867,11.254,149.471
C08826=1125.451,381.085,-87.213,-176.870,11.251,149.471
C08827=1125.455,380.838,-87.176,-176.872,11.249,149.471
C08828=1125.459,380.592,-87.139,-176.875,11.246,149.471
C08829=1125.462,380.344,-87.101,-176.879,11.244,149.471
C08830=1125.466,380.096,-87.065,-176.881,11.242,149.472
C08831=1125.470,379.850,-87.027,-176.884,11.239,149.472
C08832=1125.473,379.602,-86.990,-176.887,11.236,149.472
C08833=1125.477,379.355,-86.952,-176.890,11.235,149.472
C08834=1125.481,379.108,-86.915,-176.893,11.232,149.472
C08835=1125.485,378.861,-86.877,-176.896,11.229,149.472
C08836=1125.489,378.614,-86.841,-176.899,11.227,149.472
C08837=1125.493,378.367,-86.804,-176.902,11.225,149.472
C08838=1125.495,378.120,-86.766,-176.904,11.222,149.472
C08839=1125.499,377.872,-86.729,-176.908,11.220,149.473
C08840=1125.503,377.625,-86.693,-176.910,11.218,149.473
C08841=1125.507,377.378,-86.655,-176.913,11.215,149.473
C08842=1125.511,377.131,-86.618,-176.917,11.213,149.473
C08843=1125.515,376.884,-86.581,-176.920,11.210,149.473
C08844=1125.518,376.636,-86.544,-176.922,11.208,149.473
C08845=1125.521,376.424,-86.512,-176.925,11.206,149.474
C08846=1125.525,376.211,-86.480,-176.928,11.204,149.474
C08847=1125.528,375.999,-86.448,-176.930,11.202,149.474
C08848=1125.532,375.787,-86.416,-176.933,11.200,149.474
C08849=1125.535,375.574,-86.384,-176.935,11.198,149.474
C08850=1125.538,375.362,-86.353,-176.938,11.196,149.474
C08851=1125.541,375.149,-86.321,-176.941,11.194,149.474
C08852=1125.544,374.937,-86.289,-176.943,11.192,149.475
C08853=1125.548,374.690,-86.252,-176.947,11.189,149.475
C08854=1125.552,374.443,-86.215,-176.949,11.187,149.475
C08855=1125.555,374.195,-86.178,-176.952,11.185,149.475
C08856=1125.559,373.948,-86.141,-176.955,11.182,149.475
C08857=1125.563,373.701,-86.104,-176.959,11.180,149.475
C08858=1125.567,373.454,-86.068,-176.961,11.178,149.476
C08859=1125.571,373.206,-86.030,-176.965,11.175,149.476
C08860=1125.574,372.959,-85.994,-176.968,11.173,149.476
C08861=1125.578,372.712,-85.957,-176.971,11.171,149.476
C08862=1125.582,372.465,-85.920,-176.974,11.169,149.476
C08863=1125.586,372.218,-85.884,-176.977,11.166,149.477
C08864=1125.589,371.970,-85.847,-176.980,11.164,149.477
C08865=1125.593,371.723,-85.810,-176.983,11.161,149.477
C08866=1125.597,371.476,-85.773,-176.987,11.159,149.477
C08867=1125.601,371.229,-85.737,-176.989,11.157,149.477
C08868=1125.605,370.982,-85.700,-176.993,11.154,149.478
C08869=1125.608,370.734,-85.663,-176.996,11.152,149.478
C08870=1125.611,370.487,-85.627,-176.999,11.149,149.478
C08871=1125.616,370.240,-85.590,-177.003,11.147,149.478
C08872=1125.620,369.992,-85.553,-177.005,11.145,149.478
C08873=1125.623,369.745,-85.517,-177.009,11.143,149.479
C08874=1125.627,369.498,-85.479,-177.012,11.140,149.479
C08875=1125.631,369.250,-85.443,-177.015,11.138,149.479
C08876=1125.634,369.003,-85.407,-177.018,11.135,149.479
C08877=1125.638,368.756,-85.370,-177.022,11.133,149.479
C08878=1125.642,368.509,-85.333,-177.024,11.131,149.480
C08879=1125.646,368.262,-85.297,-177.028,11.129,149.480
C08880=1125.650,368.014,-85.260,-177.031,11.126,149.480
C08881=1125.654,367.767,-85.225,-177.034,11.124,149.480
C08882=1125.657,367.519,-85.187,-177.038,11.122,149.481
C08883=1125.661,367.272,-85.151,-177.041,11.119,149.481
C08884=1125.665,367.025,-85.114,-177.044,11.117,149.481
C08885=1125.669,366.777,-85.078,-177.047,11.115,149.481
C08886=1125.672,366.530,-85.042,-177.051,11.113,149.482
C08887=1125.676,366.283,-85.005,-177.054,11.110,149.482
C08888=1125.680,366.036,-84.969,-177.057,11.108,149.482
C08889=1125.684,365.788,-84.933,-177.061,11.105,149.482
C08890=1125.687,365.542,-84.896,-177.064,11.103,149.483
C08891=1125.692,365.294,-84.860,-177.068,11.100,149.483
C08892=1125.695,365.047,-84.824,-177.071,11.098,149.483
C08893=1125.700,364.799,-84.788,-177.074,11.096,149.483
C08894=1125.702,364.551,-84.751,-177.077,11.094,149.484
C08895=1125.707,364.304,-84.714,-177.080,11.091,149.484
C08896=1125.710,364.057,-84.679,-177.083,11.089,149.484
C08897=1125.714,363.810,-84.642,-177.087,11.087,149.484
C08898=1125.718,363.562,-84.606,-177.090,11.084,149.485
C08899=1125.722,363.315,-84.569,-177.094,11.082,149.485
C08900=1125.726,363.067,-84.534,-177.097,11.079,149.485
C08901=1125.729,362.855,-84.503,-177.100,11.078,149.485
C08902=1125.732,362.643,-84.472,-177.103,11.075,149.486
C08903=1125.735,362.430,-84.440,-177.106,11.074,149.486
C08904=1125.738,362.217,-84.409,-177.109,11.071,149.486
C08905=1125.742,362.005,-84.379,-177.112,11.069,149.486
C08906=1125.745,361.792,-84.348,-177.115,11.067,149.486
C08907=1125.749,361.580,-84.316,-177.118,11.065,149.487
C08908=1125.752,361.368,-84.286,-177.120,11.063,149.487
C08909=1125.756,361.120,-84.250,-177.124,11.061,149.487
C08910=1125.759,360.873,-84.214,-177.127,11.059,149.487
C08911=1125.764,360.625,-84.178,-177.130,11.056,149.488
C08912=1125.767,360.378,-84.142,-177.134,11.054,149.488
C08913=1125.771,360.130,-84.106,-177.137,11.052,149.488
C08914=1125.775,359.883,-84.070,-177.141,11.049,149.488
C08915=1125.779,359.636,-84.034,-177.144,11.046,149.489
C08916=1125.782,359.388,-83.999,-177.148,11.043,149.489
C08917=1125.786,359.141,-83.963,-177.151,11.041,149.489
C08918=1125.790,358.894,-83.926,-177.155,11.039,149.489
C08919=1125.794,358.646,-83.891,-177.158,11.036,149.490
C08920=1125.797,358.399,-83.855,-177.161,11.034,149.490
C08921=1125.801,358.151,-83.819,-177.165,11.032,149.490
C08922=1125.805,357.904,-83.783,-177.168,11.029,149.491
C08923=1125.809,357.657,-83.747,-177.172,11.027,149.491
C08924=1125.813,357.410,-83.712,-177.175,11.024,149.491
C08925=1125.817,357.162,-83.676,-177.179,11.022,149.491
C08926=1125.820,356.915,-83.641,-177.182,11.020,149.492
C08927=1125.825,356.667,-83.605,-177.185,11.017,149.492
C08928=1125.828,356.419,-83.569,-177.189,11.014,149.492
C08929=1125.832,356.172,-83.534,-177.193,11.012,149.492
C08930=1125.836,355.924,-83.498,-177.196,11.009,149.493
C08931=1125.840,355.677,-83.463,-177.200,11.007,149.493
C08932=1125.844,355.430,-83.427,-177.203,11.004,149.493
C08933=1125.847,355.182,-83.392,-177.207,11.002,149.493
C08934=1125.852,354.935,-83.356,-177.211,10.999,149.494
C08935=1125.855,354.687,-83.320,-177.214,10.997,149.494
C08936=1125.859,354.440,-83.284,-177.217,10.994,149.494
C08937=1125.863,354.193,-83.249,-177.221,10.992,149.495
C08938=1125.867,353.945,-83.214,-177.224,10.989,149.495
C08939=1125.871,353.698,-83.178,-177.228,10.987,149.495
C08940=1125.874,353.450,-83.143,-177.231,10.984,149.495
C08941=1125.878,353.203,-83.107,-177.235,10.981,149.495
C08942=1125.882,352.956,-83.072,-177.238,10.979,149.496
C08943=1125.886,352.709,-83.036,-177.242,10.977,149.496
C08944=1125.890,352.460,-83.002,-177.246,10.973,149.496
C08945=1125.894,352.213,-82.966,-177.249,10.971,149.496
C08946=1125.897,351.965,-82.930,-177.253,10.969,149.497
C08947=1125.902,351.719,-82.895,-177.256,10.966,149.497
C08948=1125.905,351.471,-82.860,-177.260,10.963,149.497
C08949=1125.909,351.223,-82.825,-177.263,10.961,149.497
C08950=1125.913,350.976,-82.789,-177.267,10.958,149.498
C08951=1125.917,350.729,-82.754,-177.271,10.955,149.498
C08952=1125.921,350.481,-82.719,-177.274,10.953,149.498
C08953=1125.925,350.233,-82.684,-177.278,10.950,149.499
C08954=1125.929,349.986,-82.649,-177.282,10.947,149.499
C08955=1125.933,349.739,-82.613,-177.285,10.945,149.499
C08956=1125.937,349.491,-82.578,-177.288,10.942,149.499
C08957=1125.941,349.278,-82.548,-177.291,10.940,149.499
C08958=1125.943,349.065,-82.518,-177.294,10.938,149.500
C08959=1125.947,348.853,-82.487,-177.296,10.936,149.500
C08960=1125.949,348.640,-82.457,-177.300,10.934,149.500
C08961=1125.953,348.428,-82.427,-177.302,10.932,149.500
C08962=1125.957,348.215,-82.397,-177.305,10.929,149.500
C08963=1125.960,348.002,-82.367,-177.308,10.928,149.501
C08964=1125.964,347.790,-82.337,-177.310,10.926,149.501
C08965=1125.967,347.542,-82.302,-177.314,10.923,149.501
C08966=1125.971,347.294,-82.267,-177.317,10.921,149.501
C08967=1125.975,347.047,-82.232,-177.320,10.918,149.501
C08968=1125.979,346.799,-82.197,-177.324,10.916,149.502
C08969=1125.983,346.551,-82.162,-177.327,10.913,149.502
C08970=1125.987,346.304,-82.127,-177.330,10.911,149.502
C08971=1125.990,346.057,-82.093,-177.333,10.908,149.502
C08972=1125.995,345.810,-82.057,-177.336,10.906,149.502
C08973=1125.999,345.562,-82.023,-177.340,10.903,149.502
C08974=1126.003,345.314,-81.988,-177.343,10.901,149.503
C08975=1126.006,345.067,-81.953,-177.346,10.898,149.503
C08976=1126.010,344.819,-81.918,-177.350,10.896,149.503
C08977=1126.015,344.572,-81.884,-177.353,10.893,149.503
C08978=1126.018,344.324,-81.848,-177.356,10.890,149.503
C08979=1126.022,344.076,-81.814,-177.359,10.888,149.504
C08980=1126.026,343.829,-81.780,-177.363,10.886,149.504
C08981=1126.030,343.581,-81.744,-177.366,10.883,149.504
C08982=1126.034,343.334,-81.710,-177.369,10.881,149.504
C08983=1126.038,343.086,-81.675,-177.372,10.878,149.504
C08984=1126.042,342.839,-81.641,-177.375,10.876,149.505
C08985=1126.046,342.591,-81.605,-177.378,10.874,149.505
C08986=1126.050,342.344,-81.571,-177.381,10.871,149.505
C08987=1126.054,342.096,-81.537,-177.385,10.869,149.505
C08988=1126.058,341.848,-81.502,-177.388,10.866,149.506
C08989=1126.062,341.601,-81.468,-177.391,10.864,149.506
C08990=1126.066,341.354,-81.433,-177.394,10.861,149.506
C08991=1126.070,341.106,-81.398,-177.398,10.859,149.506
C08992=1126.074,340.859,-81.364,-177.401,10.856,149.506
C08993=1126.078,340.611,-81.329,-177.404,10.854,149.507
C08994=1126.082,340.363,-81.295,-177.407,10.851,149.507
C08995=1126.085,340.115,-81.261,-177.410,10.848,149.507
C08996=1126.090,339.868,-81.226,-177.414,10.846,149.507
C08997=1126.093,339.620,-81.192,-177.417,10.844,149.507
C08998=1126.098,339.373,-81.157,-177.420,10.841,149.508
C08999=1126.101,339.125,-81.123,-177.423,10.838,149.508
C09000=1126.106,338.877,-81.089,-177.427,10.836,149.508
C09001=1126.109,338.629,-81.054,-177.430,10.833,149.508
C09002=1126.113,338.382,-81.020,-177.433,10.831,149.508
C09003=1126.117,338.134,-80.985,-177.437,10.829,149.509
C09004=1126.121,337.887,-80.951,-177.439,10.827,149.509
C09005=1126.126,337.640,-80.917,-177.442,10.824,149.509
C09006=1126.129,337.392,-80.883,-177.445,10.822,149.509
C09007=1126.133,337.144,-80.848,-177.449,10.819,149.509
C09008=1126.137,336.896,-80.814,-177.452,10.816,149.509
C09009=1126.141,336.649,-80.779,-177.455,10.814,149.510
C09010=1126.145,336.401,-80.745,-177.458,10.811,149.510
C09011=1126.148,336.154,-80.711,-177.462,10.809,149.510
C09012=1126.153,335.907,-80.677,-177.465,10.807,149.510
C09013=1126.156,335.693,-80.648,-177.467,10.805,149.511
C09014=1126.159,335.480,-80.619,-177.471,10.802,149.511
C09015=1126.163,335.268,-80.589,-177.473,10.800,149.511
C09016=1126.166,335.055,-80.560,-177.476,10.798,149.511
C09017=1126.170,334.841,-80.530,-177.478,10.796,149.511
C09018=1126.173,334.629,-80.501,-177.481,10.794,149.511
C09019=1126.176,334.416,-80.472,-177.484,10.791,149.511
C09020=1126.180,334.203,-80.443,-177.487,10.790,149.512
C09021=1126.184,333.956,-80.409,-177.490,10.787,149.512
C09022=1126.188,333.708,-80.374,-177.493,10.784,149.512
C09023=1126.192,333.461,-80.340,-177.496,10.782,149.512
C09024=1126.195,333.212,-80.307,-177.500,10.779,149.513
C09025=1126.200,332.965,-80.272,-177.503,10.777,149.513
C09026=1126.204,332.718,-80.239,-177.506,10.774,149.513
C09027=1126.207,332.469,-80.205,-177.509,10.772,149.513
C09028=1126.212,332.222,-80.171,-177.513,10.769,149.513
C09029=1126.216,331.975,-80.137,-177.515,10.766,149.513
C09030=1126.219,331.727,-80.103,-177.519,10.764,149.514
C09031=1126.224,331.479,-80.069,-177.522,10.762,149.514
C09032=1126.228,331.231,-80.036,-177.525,10.759,149.514
C09033=1126.232,330.984,-80.002,-177.528,10.756,149.514
C09034=1126.235,330.736,-79.968,-177.531,10.755,149.514
C09035=1126.240,330.488,-79.934,-177.534,10.752,149.515
C09036=1126.244,330.241,-79.900,-177.537,10.749,149.515
C09037=1126.247,329.993,-79.866,-177.541,10.747,149.515
C09038=1126.251,329.746,-79.832,-177.544,10.745,149.515
C09039=1126.255,329.498,-79.799,-177.547,10.742,149.515
C09040=1126.260,329.250,-79.765,-177.550,10.739,149.516
C09041=1126.263,329.002,-79.731,-177.553,10.737,149.516
C09042=1126.267,328.754,-79.698,-177.557,10.734,149.516
C09043=1126.271,328.507,-79.664,-177.560,10.732,149.516
C09044=1126.275,328.260,-79.631,-177.563,10.729,149.516
C09045=1126.278,328.012,-79.597,-177.566,10.727,149.517
C09046=1126.283,327.764,-79.563,-177.569,10.724,149.517
C09047=1126.288,327.516,-79.530,-177.573,10.722,149.517
C09048=1126.291,327.269,-79.496,-177.576,10.719,149.517
C09049=1126.295,327.021,-79.463,-177.579,10.717,149.517
C09050=1126.299,326.773,-79.429,-177.582,10.714,149.517
C09051=1126.303,326.526,-79.396,-177.586,10.711,149.518
C09052=1126.307,326.278,-79.362,-177.588,10.710,149.518
C09053=1126.311,326.030,-79.329,-177.591,10.707,149.518
C09054=1126.315,325.782,-79.296,-177.594,10.705,149.518
C09055=1126.319,325.534,-79.261,-177.598,10.702,149.518
C09056=1126.323,325.287,-79.228,-177.601,10.699,149.519
C09057=1126.328,325.039,-79.195,-177.604,10.697,149.519
C09058=1126.332,324.791,-79.162,-177.607,10.694,149.519
C09059=1126.336,324.543,-79.129,-177.610,10.692,149.519
C09060=1126.340,324.296,-79.095,-177.614,10.689,149.519
C09061=1126.343,324.048,-79.061,-177.617,10.687,149.520
C09062=1126.347,323.800,-79.028,-177.620,10.684,149.520
C09063=1126.351,323.552,-78.995,-177.623,10.682,149.520
C09064=1126.356,323.305,-78.962,-177.626,10.679,149.520
C09065=1126.360,323.057,-78.929,-177.629,10.676,149.520
C09066=1126.364,322.809,-78.895,-177.633,10.674,149.520
C09067=1126.367,322.562,-78.862,-177.636,10.671,149.521
C09068=1126.371,322.315,-78.829,-177.639,10.669,149.521
C09069=1126.375,322.101,-78.801,-177.642,10.667,149.521
C09070=1126.378,321.888,-78.772,-177.644,10.665,149.521
C09071=1126.382,321.675,-78.743,-177.647,10.663,149.521
C09072=1126.385,321.462,-78.715,-177.650,10.661,149.522
C09073=1126.389,321.249,-78.687,-177.652,10.659,149.522
C09074=1126.392,321.037,-78.658,-177.655,10.656,149.522
C09075=1126.396,320.823,-78.630,-177.657,10.654,149.522
C09076=1126.399,320.610,-78.601,-177.661,10.652,149.522
C09077=1126.403,320.363,-78.568,-177.664,10.649,149.522
C09078=1126.406,320.114,-78.535,-177.667,10.646,149.523
C09079=1126.410,319.867,-78.501,-177.670,10.645,149.523
C09080=1126.415,319.619,-78.468,-177.673,10.642,149.523
C09081=1126.419,319.371,-78.435,-177.676,10.640,149.523
C09082=1126.422,319.123,-78.403,-177.679,10.637,149.523
C09083=1126.427,318.875,-78.370,-177.682,10.634,149.523
C09084=1126.431,318.628,-78.337,-177.686,10.632,149.524
C09085=1126.435,318.380,-78.304,-177.689,10.629,149.524
C09086=1126.439,318.132,-78.271,-177.692,10.627,149.524
C09087=1126.442,317.885,-78.238,-177.695,10.624,149.524
C09088=1126.447,317.636,-78.206,-177.698,10.621,149.524
C09089=1126.451,317.389,-78.172,-177.701,10.619,149.525
C09090=1126.455,317.141,-78.139,-177.705,10.617,149.525
C09091=1126.459,316.893,-78.107,-177.708,10.614,149.525
C09092=1126.463,316.645,-78.074,-177.711,10.611,149.525
C09093=1126.467,316.397,-78.041,-177.714,10.609,149.525
C09094=1126.471,316.150,-78.008,-177.717,10.606,149.525
C09095=1126.475,315.902,-77.975,-177.720,10.605,149.526
C09096=1126.479,315.654,-77.943,-177.723,10.602,149.526
C09097=1126.483,315.406,-77.910,-177.726,10.599,149.526
C09098=1126.487,315.159,-77.877,-177.730,10.597,149.526
C09099=1126.491,314.910,-77.845,-177.732,10.594,149.526
C09100=1126.495,314.663,-77.812,-177.736,10.592,149.527
C09101=1126.499,314.415,-77.780,-177.739,10.589,149.527
C09102=1126.503,314.167,-77.747,-177.742,10.586,149.527
C09103=1126.508,313.920,-77.714,-177.745,10.584,149.527
C09104=1126.512,313.672,-77.682,-177.748,10.581,149.527
